C01819=1068.921,-95.321,441.532,172.288,23.007,154.216
C01820=1068.914,-95.570,441.542,172.287,23.005,154.216
C01821=1068.909,-95.820,441.552,172.285,23.004,154.216
C01822=1068.902,-96.069,441.562,172.284,23.003,154.216
C01823=1068.897,-96.318,441.573,172.282,23.001,154.216
C01824=1068.890,-96.568,441.583,172.280,23.000,154.216
C01825=1068.884,-96.818,441.594,172.279,22.999,154.216
C01826=1068.878,-97.068,441.604,172.277,22.997,154.216
C01827=1068.872,-97.318,441.614,172.275,22.996,154.216
C01828=1068.866,-97.568,441.624,172.274,22.995,154.216
C01829=1068.859,-97.850,441.635,172.272,22.993,154.215
C01830=1068.852,-98.133,441.647,172.270,22.991,154.215
C01831=1068.845,-98.416,441.659,172.268,22.990,154.215
C01832=1068.838,-98.698,441.670,172.267,22.989,154.215
C01833=1068.833,-98.948,441.681,172.265,22.987,154.215
C01834=1068.827,-99.197,441.691,172.263,22.986,154.215
C01835=1068.820,-99.447,441.701,172.261,22.985,154.215
C01836=1068.814,-99.697,441.711,172.260,22.984,154.215
C01837=1068.808,-99.947,441.722,172.258,22.982,154.215
C01838=1068.801,-100.196,441.731,172.257,22.981,154.215
C01839=1068.796,-100.446,441.742,172.255,22.980,154.215
C01840=1068.789,-100.696,441.752,172.253,22.978,154.215
C01841=1068.783,-100.945,441.761,172.252,22.977,154.215
C01842=1068.777,-101.195,441.771,172.250,22.976,154.215
C01843=1068.771,-101.445,441.782,172.248,22.975,154.215
C01844=1068.764,-101.695,441.792,172.247,22.974,154.215
C01845=1068.758,-101.944,441.802,172.245,22.972,154.215
C01846=1068.753,-102.194,441.812,172.243,22.971,154.215
C01847=1068.746,-102.444,441.822,172.242,22.970,154.215
C01848=1068.740,-102.693,441.832,172.240,22.968,154.215
C01849=1068.734,-102.943,441.843,172.238,22.968,154.216
C01850=1068.728,-103.193,441.852,172.237,22.966,154.215
C01851=1068.722,-103.443,441.862,172.235,22.965,154.215
C01852=1068.716,-103.692,441.873,172.234,22.964,154.215
C01853=1068.710,-103.942,441.882,172.232,22.962,154.215
C01854=1068.704,-104.192,441.892,172.230,22.961,154.215
C01855=1068.697,-104.441,441.902,172.228,22.960,154.216
C01856=1068.692,-104.691,441.912,172.227,22.959,154.216
C01857=1068.686,-104.941,441.922,172.225,22.958,154.216
C01858=1068.680,-105.191,441.931,172.224,22.956,154.216
C01859=1068.673,-105.440,441.942,172.222,22.956,154.216
C01860=1068.667,-105.691,441.952,172.220,22.954,154.216
C01861=1068.661,-105.940,441.962,172.219,22.953,154.216
C01862=1068.654,-106.189,441.972,172.217,22.952,154.216
C01863=1068.648,-106.439,441.982,172.215,22.951,154.216
C01864=1068.643,-106.689,441.992,172.213,22.949,154.216
C01865=1068.637,-106.939,442.001,172.212,22.948,154.216
C01866=1068.630,-107.188,442.012,172.210,22.947,154.216
C01867=1068.624,-107.438,442.021,172.208,22.946,154.216
C01868=1068.618,-107.688,442.031,172.207,22.945,154.216
C01869=1068.612,-107.938,442.041,172.205,22.943,154.216
C01870=1068.606,-108.188,442.051,172.203,22.943,154.216
C01871=1068.600,-108.437,442.061,172.202,22.941,154.216
C01872=1068.594,-108.687,442.070,172.200,22.940,154.216
C01873=1068.587,-108.937,442.080,172.198,22.939,154.216
C01874=1068.581,-109.186,442.090,172.197,22.938,154.216
C01875=1068.575,-109.436,442.099,172.195,22.937,154.216
C01876=1068.569,-109.685,442.109,172.193,22.936,154.216
C01877=1068.562,-109.935,442.119,172.191,22.935,154.216
C01878=1068.557,-110.185,442.129,172.190,22.934,154.216
C01879=1068.551,-110.435,442.139,172.188,22.932,154.216
C01880=1068.545,-110.685,442.148,172.187,22.932,154.216
C01881=1068.539,-110.935,442.158,172.186,22.931,154.216
C01882=1068.532,-111.185,442.167,172.184,22.930,154.216
C01883=1068.526,-111.434,442.178,172.182,22.929,154.216
C01884=1068.520,-111.683,442.187,172.181,22.928,154.216
C01885=1068.514,-111.933,442.197,172.179,22.926,154.216
C01886=1068.507,-112.183,442.206,172.177,22.925,154.216
C01887=1068.501,-112.433,442.216,172.175,22.924,154.216
C01888=1068.495,-112.683,442.226,172.174,22.923,154.216
C01889=1068.490,-112.933,442.236,172.172,22.922,154.217
C01890=1068.483,-113.183,442.245,172.170,22.921,154.217
C01891=1068.478,-113.432,442.254,172.169,22.920,154.217
C01892=1068.472,-113.681,442.264,172.167,22.919,154.217
C01893=1068.465,-113.962,442.275,172.165,22.918,154.217
C01894=1068.458,-114.243,442.286,172.163,22.916,154.217
C01895=1068.450,-114.522,442.296,172.161,22.916,154.217
C01896=1068.443,-114.803,442.307,172.159,22.914,154.217
C01897=1068.437,-115.053,442.317,172.157,22.913,154.217
C01898=1068.431,-115.303,442.326,172.156,22.912,154.217
C01899=1068.425,-115.552,442.336,172.154,22.911,154.217
C01900=1068.419,-115.802,442.346,172.152,22.910,154.217
C01901=1068.413,-116.052,442.355,172.151,22.909,154.217
C01902=1068.406,-116.302,442.365,172.149,22.909,154.217
C01903=1068.400,-116.552,442.374,172.147,22.907,154.217
C01904=1068.395,-116.801,442.384,172.145,22.906,154.217
C01905=1068.389,-117.050,442.393,172.144,22.906,154.218
C01906=1068.382,-117.300,442.403,172.143,22.905,154.217
C01907=1068.376,-117.550,442.412,172.141,22.904,154.218
C01908=1068.370,-117.800,442.422,172.139,22.903,154.218
C01909=1068.364,-118.050,442.431,172.138,22.902,154.218
C01910=1068.358,-118.300,442.440,172.136,22.901,154.218
C01911=1068.351,-118.550,442.449,172.134,22.900,154.218
C01912=1068.345,-118.799,442.459,172.132,22.899,154.218
C01913=1068.339,-119.049,442.468,172.131,22.898,154.218
C01914=1068.333,-119.298,442.478,172.129,22.897,154.218
C01915=1068.327,-119.548,442.487,172.127,22.896,154.218
C01916=1068.321,-119.798,442.497,172.125,22.895,154.218
C01917=1068.315,-120.048,442.506,172.124,22.895,154.218
C01918=1068.308,-120.297,442.516,172.122,22.893,154.218
C01919=1068.303,-120.548,442.525,172.120,22.893,154.218
C01920=1068.296,-120.798,442.534,172.118,22.892,154.219
C01921=1068.289,-121.047,442.543,172.117,22.890,154.219
C01922=1068.284,-121.296,442.552,172.115,22.890,154.219
C01923=1068.278,-121.546,442.562,172.113,22.889,154.219
C01924=1068.272,-121.796,442.572,172.111,22.888,154.219
C01925=1068.265,-122.046,442.581,172.110,22.887,154.219
C01926=1068.260,-122.296,442.590,172.109,22.886,154.219
C01927=1068.253,-122.546,442.599,172.107,22.886,154.219
C01928=1068.247,-122.795,442.608,172.105,22.885,154.219
C01929=1068.241,-123.044,442.618,172.103,22.884,154.219
C01930=1068.235,-123.294,442.627,172.102,22.883,154.219
C01931=1068.229,-123.545,442.636,172.100,22.882,154.219
C01932=1068.223,-123.794,442.646,172.098,22.881,154.219
C01933=1068.217,-124.044,442.655,172.096,22.880,154.220
C01934=1068.210,-124.293,442.664,172.095,22.880,154.220
C01935=1068.204,-124.543,442.673,172.093,22.879,154.220
C01936=1068.198,-124.793,442.682,172.091,22.878,154.220
C01937=1068.192,-125.043,442.692,172.089,22.877,154.220
C01938=1068.185,-125.292,442.701,172.088,22.876,154.220
C01939=1068.180,-125.542,442.709,172.086,22.875,154.220
C01940=1068.174,-125.792,442.719,172.084,22.875,154.220
C01941=1068.167,-126.042,442.728,172.083,22.874,154.220
C01942=1068.161,-126.291,442.737,172.081,22.873,154.220
C01943=1068.155,-126.542,442.746,172.079,22.873,154.221
C01944=1068.149,-126.791,442.756,172.078,22.872,154.221
C01945=1068.142,-127.040,442.764,172.076,22.871,154.221
C01946=1068.136,-127.291,442.773,172.074,22.870,154.221
C01947=1068.130,-127.540,442.783,172.072,22.870,154.221
C01948=1068.124,-127.790,442.792,172.070,22.869,154.221
C01949=1068.118,-128.041,442.801,172.069,22.868,154.221
C01950=1068.115,-128.291,442.812,172.067,22.866,154.221
C01951=1068.113,-128.542,442.822,172.066,22.863,154.221
C01952=1068.113,-128.793,442.834,172.065,22.860,154.220
C01953=1068.115,-129.046,442.847,172.064,22.856,154.220
C01954=1068.119,-129.298,442.860,172.064,22.852,154.219
C01955=1068.125,-129.549,442.875,172.064,22.847,154.218
C01956=1068.132,-129.799,442.890,172.064,22.841,154.217
C01957=1067.743,-129.822,442.718,172.016,22.987,154.250
C01958=1067.737,-129.572,442.703,172.017,22.993,154.251
C01959=1067.732,-129.320,442.688,172.017,22.997,154.252
C01960=1067.727,-129.068,442.675,172.018,23.002,154.252
C01961=1067.725,-128.816,442.662,172.018,23.005,154.253
C01962=1067.725,-128.565,442.650,172.019,23.009,154.254
C01963=1067.726,-128.314,442.639,172.020,23.011,154.254
C01964=1067.730,-128.063,442.629,172.021,23.013,154.254
C01965=1067.736,-127.812,442.619,172.023,23.014,154.254
C01966=1067.742,-127.563,442.610,172.025,23.015,154.254
C01967=1067.747,-127.313,442.601,172.027,23.015,154.254
C01968=1067.754,-127.063,442.592,172.029,23.016,154.254
C01969=1067.760,-126.814,442.583,172.030,23.017,154.253
C01970=1067.766,-126.564,442.573,172.032,23.018,154.253
C01971=1067.773,-126.314,442.564,172.034,23.018,154.253
C01972=1067.778,-126.065,442.556,172.036,23.019,154.253
C01973=1067.785,-125.815,442.546,172.037,23.021,154.253
C01974=1067.791,-125.565,442.537,172.039,23.021,154.253
C01975=1067.797,-125.315,442.528,172.040,23.022,154.253
C01976=1067.804,-125.065,442.519,172.042,23.022,154.253
C01977=1067.810,-124.815,442.509,172.044,23.023,154.253
C01978=1067.815,-124.566,442.500,172.045,23.024,154.253
C01979=1067.822,-124.316,442.492,172.047,23.025,154.252
C01980=1067.828,-124.066,442.482,172.049,23.025,154.252
C01981=1067.834,-123.816,442.473,172.051,23.027,154.252
C01982=1067.840,-123.567,442.463,172.053,23.028,154.252
C01983=1067.846,-123.317,442.455,172.054,23.028,154.252
C01984=1067.852,-123.067,442.445,172.056,23.029,154.252
C01985=1067.859,-122.818,442.436,172.058,23.030,154.252
C01986=1067.865,-122.568,442.427,172.060,23.031,154.252
C01987=1067.871,-122.318,442.417,172.061,23.032,154.252
C01988=1067.877,-122.068,442.407,172.063,23.033,154.252
C01989=1067.883,-121.819,442.399,172.065,23.033,154.252
C01990=1067.889,-121.569,442.389,172.067,23.034,154.251
C01991=1067.896,-121.319,442.380,172.068,23.035,154.251
C01992=1067.902,-121.069,442.371,172.070,23.036,154.251
C01993=1067.908,-120.820,442.361,172.071,23.037,154.251
C01994=1067.914,-120.570,442.352,172.073,23.038,154.251
C01995=1067.920,-120.319,442.343,172.075,23.039,154.251
C01996=1067.926,-120.070,442.334,172.076,23.039,154.251
C01997=1067.932,-119.821,442.324,172.078,23.040,154.251
C01998=1067.938,-119.571,442.315,172.080,23.042,154.251
C01999=1067.944,-119.321,442.305,172.082,23.042,154.251
C02000=1067.951,-119.071,442.296,172.083,23.043,154.251
C02001=1067.957,-118.822,442.286,172.085,23.044,154.251
C02002=1067.963,-118.572,442.277,172.087,23.045,154.251
C02003=1067.970,-118.322,442.267,172.089,23.046,154.251
C02004=1067.976,-118.072,442.258,172.090,23.047,154.251
C02005=1067.981,-117.823,442.249,172.092,23.048,154.250
C02006=1067.987,-117.573,442.240,172.094,23.049,154.250
C02007=1067.993,-117.323,442.230,172.095,23.050,154.250
C02008=1067.999,-117.073,442.221,172.097,23.051,154.250
C02009=1068.006,-116.823,442.211,172.099,23.052,154.250
C02010=1068.012,-116.574,442.201,172.101,23.053,154.250
C02011=1068.018,-116.324,442.192,172.103,23.054,154.250
C02012=1068.024,-116.074,442.182,172.104,23.055,154.250
C02013=1068.030,-115.824,442.173,172.106,23.056,154.250
C02014=1068.037,-115.574,442.163,172.108,23.056,154.250
C02015=1068.043,-115.325,442.154,172.109,23.058,154.250
C02016=1068.049,-115.075,442.144,172.110,23.058,154.250
C02017=1068.054,-114.826,442.135,172.112,23.059,154.250
C02018=1068.062,-114.545,442.124,172.115,23.061,154.250
C02019=1068.069,-114.265,442.113,172.116,23.062,154.250
C02020=1068.076,-113.984,442.102,172.118,23.063,154.249
C02021=1068.083,-113.703,442.092,172.120,23.064,154.250
C02022=1068.089,-113.453,442.082,172.122,23.065,154.249
C02023=1068.095,-113.205,442.072,172.123,23.066,154.249
C02024=1068.101,-112.955,442.063,172.125,23.067,154.249
C02025=1068.107,-112.705,442.053,172.127,23.068,154.249
C02026=1068.113,-112.455,442.043,172.128,23.069,154.249
C02027=1068.119,-112.205,442.033,172.130,23.070,154.249
C02028=1068.125,-111.955,442.024,172.132,23.072,154.249
C02029=1068.131,-111.706,442.014,172.133,23.072,154.249
C02030=1068.137,-111.456,442.005,172.135,23.074,154.249
C02031=1068.144,-111.206,441.995,172.137,23.074,154.249
C02032=1068.150,-110.956,441.986,172.139,23.076,154.249
C02033=1068.156,-110.707,441.975,172.140,23.076,154.249
C02034=1068.162,-110.457,441.966,172.142,23.078,154.249
C02035=1068.169,-110.207,441.956,172.144,23.079,154.249
C02036=1068.175,-109.958,441.947,172.145,23.080,154.249
C02037=1068.180,-109.707,441.937,172.147,23.081,154.249
C02038=1068.186,-109.458,441.927,172.149,23.082,154.249
C02039=1068.193,-109.208,441.917,172.150,23.083,154.249
C02040=1068.199,-108.959,441.907,172.152,23.085,154.249
C02041=1068.205,-108.709,441.898,172.154,23.085,154.249
C02042=1068.211,-108.459,441.888,172.155,23.087,154.249
C02043=1068.218,-108.209,441.878,172.157,23.087,154.249
C02044=1068.224,-107.960,441.868,172.159,23.089,154.249
C02045=1068.229,-107.710,441.858,172.161,23.090,154.249
C02046=1068.236,-107.460,441.848,172.162,23.091,154.248
C02047=1068.242,-107.210,441.839,172.164,23.092,154.248
C02048=1068.248,-106.961,441.829,172.166,23.093,154.248
C02049=1068.254,-106.711,441.819,172.167,23.094,154.248
C02050=1068.260,-106.461,441.809,172.169,23.096,154.248
C02051=1068.266,-106.212,441.799,172.171,23.097,154.248
C02052=1068.273,-105.962,441.789,172.172,23.098,154.248
C02053=1068.279,-105.713,441.779,172.174,23.099,154.248
C02054=1068.285,-105.462,441.769,172.176,23.100,154.248
C02055=1068.291,-105.212,441.759,172.177,23.102,154.248
C02056=1068.297,-104.963,441.749,172.179,23.103,154.248
C02057=1068.304,-104.713,441.739,172.181,23.104,154.248
C02058=1068.309,-104.463,441.729,172.182,23.105,154.248
C02059=1068.315,-104.214,441.719,172.184,23.106,154.248
C02060=1068.322,-103.964,441.709,172.185,23.107,154.248
C02061=1068.328,-103.714,441.700,172.186,23.109,154.248
C02062=1068.334,-103.465,441.689,172.188,23.109,154.248
C02063=1068.340,-103.215,441.679,172.190,23.111,154.248
C02064=1068.346,-102.965,441.670,172.192,23.112,154.248
C02065=1068.352,-102.715,441.659,172.193,23.113,154.248
C02066=1068.358,-102.466,441.649,172.195,23.115,154.248
C02067=1068.364,-102.216,441.640,172.196,23.116,154.248
C02068=1068.370,-101.967,441.630,172.198,23.117,154.248
C02069=1068.376,-101.717,441.619,172.200,23.118,154.248
C02070=1068.383,-101.467,441.609,172.201,23.119,154.248
C02071=1068.389,-101.217,441.599,172.203,23.121,154.248
C02072=1068.395,-100.967,441.589,172.205,23.122,154.248
C02073=1068.401,-100.718,441.579,172.206,23.123,154.248
C02074=1068.407,-100.468,441.569,172.208,23.125,154.248
C02075=1068.413,-100.218,441.558,172.210,23.126,154.248
C02076=1068.419,-99.969,441.549,172.211,23.127,154.248
C02077=1068.426,-99.719,441.538,172.213,23.128,154.248
C02078=1068.432,-99.469,441.528,172.215,23.129,154.248
C02079=1068.438,-99.219,441.518,172.216,23.131,154.248
C02080=1068.444,-98.970,441.508,172.218,23.132,154.248
C02081=1068.450,-98.719,441.498,172.220,23.133,154.248
C02082=1068.457,-98.436,441.486,172.222,23.135,154.248
C02083=1068.464,-98.154,441.475,172.224,23.136,154.248
C02084=1068.471,-97.871,441.463,172.225,23.138,154.248
C02085=1068.477,-97.589,441.452,172.227,23.139,154.248
C02086=1068.484,-97.339,441.441,172.230,23.141,154.248
C02087=1068.490,-97.089,441.431,172.231,23.142,154.248
C02088=1068.496,-96.840,441.421,172.233,23.143,154.248
C02089=1068.502,-96.590,441.410,172.234,23.145,154.248
C02090=1068.508,-96.341,441.400,172.236,23.147,154.248
C02091=1068.514,-96.091,441.389,172.238,23.148,154.248
C02092=1068.520,-95.841,441.380,172.239,23.149,154.248
C02093=1068.526,-95.592,441.369,172.241,23.150,154.248
C02094=1068.532,-95.341,441.359,172.242,23.152,154.248
C02095=1068.538,-95.092,441.348,172.244,23.153,154.249
C02096=1068.544,-94.842,441.337,172.246,23.154,154.249
C02097=1068.550,-94.592,441.328,172.247,23.156,154.249
C02098=1068.556,-94.343,441.317,172.249,23.157,154.249
C02099=1068.562,-94.093,441.307,172.250,23.159,154.249
C02100=1068.568,-93.844,441.296,172.252,23.160,154.249
C02101=1068.575,-93.594,441.286,172.254,23.162,154.249
C02102=1068.580,-93.344,441.276,172.255,23.163,154.249
C02103=1068.586,-93.094,441.265,172.257,23.164,154.249
C02104=1068.592,-92.844,441.255,172.259,23.166,154.249
C02105=1068.598,-92.595,441.244,172.260,23.167,154.249
C02106=1068.605,-92.345,441.234,172.262,23.169,154.249
C02107=1068.611,-92.095,441.224,172.263,23.170,154.249
C02108=1068.616,-91.845,441.213,172.265,23.171,154.249
C02109=1068.623,-91.596,441.202,172.267,23.173,154.249
C02110=1068.629,-91.347,441.191,172.268,23.174,154.249
C02111=1068.635,-91.096,441.182,172.270,23.176,154.249
C02112=1068.641,-90.847,441.171,172.271,23.177,154.249
C02113=1068.647,-90.597,441.160,172.273,23.179,154.249
C02114=1068.653,-90.347,441.150,172.275,23.180,154.249
C02115=1068.659,-90.098,441.139,172.276,23.181,154.249
C02116=1068.666,-89.848,441.129,172.278,23.183,154.249
C02117=1068.671,-89.599,441.118,172.279,23.184,154.249
C02118=1068.677,-89.349,441.108,172.281,23.186,154.249
C02119=1068.683,-89.099,441.097,172.283,23.187,154.249
C02120=1068.690,-88.849,441.086,172.284,23.189,154.250
C02121=1068.696,-88.600,441.076,172.286,23.190,154.250
C02122=1068.702,-88.350,441.066,172.287,23.192,154.250
C02123=1068.707,-88.100,441.055,172.289,23.193,154.250
C02124=1068.714,-87.850,441.044,172.290,23.195,154.250
C02125=1068.720,-87.601,441.033,172.292,23.196,154.250
C02126=1068.726,-87.352,441.022,172.294,23.197,154.250
C02127=1068.733,-87.101,441.012,172.295,23.199,154.250
C02128=1068.738,-86.852,441.002,172.297,23.201,154.250
C02129=1068.744,-86.602,440.991,172.298,23.202,154.250
C02130=1068.751,-86.353,440.980,172.300,23.203,154.250
C02131=1068.757,-86.103,440.969,172.301,23.205,154.250
C02132=1068.762,-85.853,440.959,172.303,23.206,154.250
C02133=1068.769,-85.603,440.949,172.305,23.208,154.250
C02134=1068.775,-85.353,440.938,172.306,23.209,154.250
C02135=1068.781,-85.104,440.927,172.308,23.211,154.250
C02136=1068.787,-84.855,440.916,172.309,23.212,154.250
C02137=1068.794,-84.604,440.905,172.311,23.214,154.250
C02138=1068.800,-84.355,440.894,172.313,23.215,154.250
C02139=1068.806,-84.106,440.884,172.314,23.217,154.250
C02140=1068.812,-83.855,440.873,172.316,23.218,154.251
C02141=1068.818,-83.605,440.863,172.317,23.220,154.251
C02142=1068.824,-83.356,440.852,172.320,23.222,154.251
C02143=1068.831,-83.106,440.841,172.321,23.223,154.251
C02144=1068.836,-82.856,440.830,172.323,23.225,154.251
C02145=1068.843,-82.607,440.820,172.325,23.226,154.251
C02146=1068.850,-82.326,440.807,172.326,23.228,154.251
C02147=1068.857,-82.046,440.795,172.328,23.229,154.251
C02148=1068.864,-81.766,440.783,172.329,23.231,154.251
C02149=1068.871,-81.486,440.771,172.332,23.233,154.251
C02150=1068.877,-81.235,440.759,172.333,23.235,154.251
C02151=1068.883,-80.986,440.749,172.335,23.236,154.251
C02152=1068.889,-80.737,440.738,172.336,23.238,154.251
C02153=1068.895,-80.487,440.727,172.338,23.239,154.251
C02154=1068.902,-80.237,440.717,172.339,23.241,154.251
C02155=1068.908,-79.987,440.705,172.341,23.243,154.252
C02156=1068.914,-79.738,440.694,172.343,23.244,154.252
C02157=1068.920,-79.488,440.684,172.344,23.246,154.252
C02158=1068.926,-79.238,440.672,172.346,23.247,154.252
C02159=1068.932,-78.989,440.661,172.347,23.249,154.252
C02160=1068.938,-78.739,440.651,172.349,23.250,154.252
C02161=1068.945,-78.489,440.640,172.350,23.252,154.252
C02162=1068.950,-78.240,440.629,172.352,23.254,154.252
C02163=1068.957,-77.990,440.618,172.353,23.255,154.252
C02164=1068.962,-77.740,440.607,172.355,23.257,154.252
C02165=1068.968,-77.491,440.596,172.356,23.259,154.252
C02166=1068.975,-77.240,440.585,172.358,23.260,154.253
C02167=1068.980,-76.991,440.574,172.360,23.262,154.253
C02168=1068.986,-76.741,440.563,172.361,23.264,154.253
C02169=1068.993,-76.492,440.551,172.363,23.266,154.253
C02170=1068.998,-76.242,440.540,172.365,23.267,154.253
C02171=1069.005,-75.992,440.529,172.366,23.269,154.253
C02172=1069.010,-75.743,440.518,172.368,23.270,154.253
C02173=1069.017,-75.492,440.507,172.370,23.272,154.253
C02174=1069.023,-75.243,440.497,172.371,23.274,154.253
C02175=1069.029,-74.994,440.486,172.373,23.275,154.253
C02176=1069.036,-74.744,440.474,172.374,23.277,154.253
C02177=1069.041,-74.495,440.463,172.376,23.279,154.253
C02178=1069.048,-74.245,440.452,172.377,23.281,154.254
C02179=1069.054,-73.995,440.441,172.379,23.282,154.254
C02180=1069.060,-73.745,440.430,172.380,23.284,154.254
C02181=1069.066,-73.496,440.418,172.382,23.286,154.254
C02182=1069.071,-73.246,440.406,172.383,23.287,154.254
C02183=1069.077,-72.996,440.395,172.385,23.289,154.254
C02184=1069.083,-72.747,440.384,172.386,23.291,154.254
C02185=1069.089,-72.496,440.373,172.388,23.293,154.254
C02186=1069.095,-72.247,440.362,172.389,23.294,154.254
C02187=1069.101,-71.998,440.351,172.391,23.296,154.255
C02188=1069.107,-71.747,440.339,172.392,23.298,154.255
C02189=1069.112,-71.498,440.328,172.394,23.299,154.255
C02190=1069.119,-71.248,440.316,172.395,23.301,154.255
C02191=1069.125,-70.999,440.305,172.397,23.303,154.255
C02192=1069.131,-70.749,440.294,172.399,23.305,154.255
C02193=1069.137,-70.500,440.282,172.401,23.307,154.255
C02194=1069.142,-70.250,440.271,172.402,23.309,154.255
C02195=1069.149,-70.000,440.260,172.404,23.311,154.255
C02196=1069.155,-69.751,440.248,172.405,23.312,154.256
C02197=1069.161,-69.501,440.237,172.407,23.314,154.256
C02198=1069.167,-69.251,440.226,172.408,23.316,154.256
C02199=1069.173,-69.002,440.214,172.410,23.318,154.256
C02200=1069.178,-68.752,440.202,172.411,23.320,154.256
C02201=1069.185,-68.502,440.191,172.413,23.321,154.256
C02202=1069.191,-68.253,440.180,172.414,23.323,154.256
C02203=1069.197,-68.003,440.168,172.416,23.325,154.256
C02204=1069.203,-67.753,440.157,172.417,23.327,154.257
C02205=1069.209,-67.503,440.145,172.419,23.329,154.257
C02206=1069.214,-67.254,440.134,172.420,23.331,154.257
C02207=1069.221,-67.004,440.122,172.421,23.333,154.257
C02208=1069.227,-66.755,440.111,172.423,23.334,154.257
C02209=1069.232,-66.504,440.099,172.425,23.336,154.257
C02210=1069.239,-66.227,440.087,172.427,23.339,154.257
C02211=1069.246,-65.949,440.073,172.428,23.340,154.258
C02212=1069.253,-65.670,440.061,172.430,23.342,154.258
C02213=1069.259,-65.392,440.048,172.432,23.345,154.258
C02214=1069.265,-65.142,440.037,172.434,23.346,154.258
C02215=1069.272,-64.893,440.025,172.435,23.348,154.258
C02216=1069.278,-64.643,440.014,172.436,23.350,154.258
C02217=1069.283,-64.393,440.002,172.438,23.352,154.258
C02218=1069.289,-64.144,439.991,172.440,23.353,154.258
C02219=1069.296,-63.894,439.979,172.441,23.355,154.259
C02220=1069.302,-63.645,439.968,172.443,23.357,154.259
C02221=1069.307,-63.395,439.955,172.444,23.359,154.259
C02222=1069.314,-63.145,439.944,172.445,23.361,154.259
C02223=1069.320,-62.896,439.932,172.447,23.363,154.259
C02224=1069.326,-62.645,439.921,172.448,23.365,154.259
C02225=1069.332,-62.396,439.909,172.450,23.366,154.259
C02226=1069.338,-62.146,439.898,172.451,23.368,154.260
C02227=1069.345,-61.897,439.886,172.453,23.370,154.260
C02228=1069.350,-61.647,439.874,172.454,23.372,154.260
C02229=1069.356,-61.397,439.862,172.456,23.374,154.260
C02230=1069.362,-61.148,439.851,172.458,23.376,154.260
C02231=1069.369,-60.898,439.840,172.460,23.378,154.260
C02232=1069.374,-60.648,439.827,172.461,23.380,154.260
C02233=1069.380,-60.399,439.816,172.463,23.382,154.261
C02234=1069.387,-60.149,439.804,172.464,23.384,154.261
C02235=1069.392,-59.900,439.792,172.465,23.386,154.261
C02236=1069.398,-59.650,439.781,172.467,23.387,154.261
C02237=1069.405,-59.400,439.769,172.468,23.389,154.261
C02238=1069.411,-59.151,439.758,172.470,23.391,154.261
C02239=1069.417,-58.901,439.745,172.471,23.393,154.261
C02240=1069.423,-58.651,439.733,172.473,23.395,154.262
C02241=1069.429,-58.402,439.722,172.474,23.397,154.262
C02242=1069.435,-58.152,439.710,172.476,23.399,154.262
C02243=1069.442,-57.902,439.698,172.477,23.400,154.262
C02244=1069.447,-57.653,439.687,172.479,23.402,154.262
C02245=1069.453,-57.403,439.675,172.480,23.404,154.262
C02246=1069.460,-57.153,439.663,172.482,23.406,154.263
C02247=1069.466,-56.904,439.652,172.484,23.408,154.263
C02248=1069.472,-56.654,439.639,172.485,23.410,154.263
C02249=1069.478,-56.404,439.627,172.487,23.412,154.263
C02250=1069.485,-56.155,439.615,172.488,23.414,154.263
C02251=1069.490,-55.905,439.604,172.490,23.416,154.263
C02252=1069.497,-55.655,439.592,172.491,23.418,154.263
C02253=1069.503,-55.406,439.580,172.493,23.420,154.263
C02254=1069.509,-55.157,439.568,172.494,23.421,154.264
C02255=1069.515,-54.907,439.556,172.496,23.423,154.264
C02256=1069.522,-54.657,439.544,172.497,23.425,154.264
C02257=1069.527,-54.407,439.532,172.499,23.428,154.264
C02258=1069.534,-54.158,439.520,172.500,23.429,154.264
C02259=1069.540,-53.908,439.509,172.502,23.431,154.264
C02260=1069.546,-53.658,439.496,172.503,23.433,154.265
C02261=1069.552,-53.409,439.485,172.504,23.435,154.265
C02262=1069.558,-53.160,439.473,172.507,23.437,154.265
C02263=1069.564,-52.910,439.460,172.508,23.439,154.265
C02264=1069.571,-52.660,439.449,172.510,23.441,154.265
C02265=1069.577,-52.410,439.437,172.511,23.443,154.265
C02266=1069.583,-52.161,439.425,172.513,23.445,154.265
C02267=1069.589,-51.911,439.413,172.514,23.447,154.266
C02268=1069.595,-51.661,439.400,172.516,23.449,154.266
C02269=1069.602,-51.412,439.389,172.517,23.451,154.266
C02270=1069.608,-51.162,439.376,172.518,23.453,154.266
C02271=1069.613,-50.912,439.365,172.520,23.455,154.266
C02272=1069.620,-50.663,439.353,172.521,23.457,154.266
C02273=1069.626,-50.413,439.341,172.523,23.458,154.267
C02274=1069.633,-50.136,439.327,172.525,23.461,154.267
C02275=1069.639,-49.859,439.314,172.527,23.463,154.267
C02276=1069.646,-49.583,439.300,172.528,23.466,154.267
C02277=1069.653,-49.306,439.287,172.529,23.467,154.267
C02278=1069.659,-49.056,439.274,172.532,23.470,154.268
C02279=1069.665,-48.806,439.262,172.533,23.472,154.268
C02280=1069.671,-48.557,439.250,172.534,23.474,154.268
C02281=1069.677,-48.307,439.237,172.536,23.476,154.268
C02282=1069.683,-48.058,439.225,172.537,23.478,154.268
C02283=1069.689,-47.808,439.213,172.539,23.480,154.269
C02284=1069.694,-47.558,439.201,172.540,23.483,154.269
C02285=1069.701,-47.309,439.189,172.542,23.484,154.269
C02286=1069.707,-47.059,439.176,172.543,23.486,154.269
C02287=1069.713,-46.809,439.164,172.544,23.489,154.269
C02288=1069.719,-46.560,439.152,172.546,23.491,154.270
C02289=1069.725,-46.310,439.139,172.547,23.492,154.270
C02290=1069.731,-46.060,439.127,172.549,23.495,154.270
C02291=1069.737,-45.811,439.115,172.550,23.497,154.270
C02292=1069.743,-45.561,439.102,172.552,23.499,154.270
C02293=1069.749,-45.312,439.090,172.554,23.501,154.270
C02294=1069.755,-45.062,439.078,172.555,23.503,154.271
C02295=1069.761,-44.812,439.066,172.557,23.505,154.271
C02296=1069.767,-44.562,439.053,172.558,23.508,154.271
C02297=1069.773,-44.313,439.041,172.559,23.509,154.271
C02298=1069.779,-44.064,439.029,172.561,23.512,154.271
C02299=1069.785,-43.814,439.016,172.562,23.514,154.272
C02300=1069.791,-43.564,439.004,172.564,23.516,154.272
C02301=1069.797,-43.314,438.991,172.565,23.518,154.272
C02302=1069.803,-43.065,438.979,172.567,23.520,154.272
C02303=1069.810,-42.815,438.966,172.568,23.522,154.272
C02304=1069.815,-42.566,438.954,172.569,23.524,154.273
C02305=1069.821,-42.316,438.941,172.571,23.526,154.273
C02306=1069.827,-42.067,438.929,172.572,23.528,154.273
C02307=1069.833,-41.817,438.917,172.574,23.531,154.273
C02308=1069.839,-41.567,438.904,172.576,23.533,154.273
C02309=1069.846,-41.317,438.892,172.577,23.535,154.274
C02310=1069.852,-41.068,438.879,172.579,23.537,154.274
C02311=1069.858,-40.818,438.866,172.580,23.539,154.274
C02312=1069.863,-40.569,438.854,172.582,23.541,154.274
C02313=1069.870,-40.319,438.842,172.583,23.543,154.274
C02314=1069.876,-40.069,438.830,172.584,23.545,154.275
C02315=1069.882,-39.820,438.816,172.586,23.547,154.275
C02316=1069.888,-39.570,438.804,172.587,23.550,154.275
C02317=1069.894,-39.320,438.791,172.589,23.552,154.275
C02318=1069.901,-39.071,438.779,172.590,23.554,154.275
C02319=1069.907,-38.821,438.767,172.591,23.556,154.276
C02320=1069.913,-38.572,438.754,172.593,23.558,154.276
C02321=1069.919,-38.322,438.741,172.595,23.560,154.276
C02322=1069.924,-38.073,438.729,172.596,23.563,154.276
C02323=1069.930,-37.823,438.716,172.598,23.565,154.276
C02324=1069.936,-37.574,438.703,172.599,23.567,154.277
C02325=1069.942,-37.324,438.690,172.601,23.569,154.277
C02326=1069.948,-37.074,438.678,172.602,23.571,154.277
C02327=1069.954,-36.825,438.665,172.603,23.573,154.277
C02328=1069.961,-36.575,438.653,172.605,23.576,154.277
C02329=1069.967,-36.325,438.640,172.606,23.578,154.278
C02330=1069.973,-36.076,438.627,172.608,23.580,154.278
C02331=1069.978,-35.827,438.615,172.609,23.582,154.278
C02332=1069.984,-35.577,438.602,172.610,23.584,154.278
C02333=1069.990,-35.327,438.589,172.612,23.587,154.279
C02334=1069.996,-35.078,438.576,172.613,23.589,154.279
C02335=1070.002,-34.828,438.564,172.615,23.591,154.279
C02336=1070.008,-34.578,438.550,172.617,23.594,154.279
C02337=1070.014,-34.329,438.538,172.618,23.596,154.279
C02338=1070.021,-34.052,438.523,172.619,23.598,154.280
C02339=1070.027,-33.775,438.510,172.621,23.601,154.280
C02340=1070.034,-33.499,438.495,172.623,23.603,154.280
C02341=1070.040,-33.222,438.481,172.624,23.606,154.280
C02342=1070.046,-32.973,438.468,172.626,23.608,154.281
C02343=1070.053,-32.723,438.455,172.627,23.610,154.281
C02344=1070.058,-32.473,438.442,172.629,23.612,154.281
C02345=1070.064,-32.223,438.430,172.630,23.614,154.281
C02346=1070.071,-31.974,438.416,172.631,23.617,154.282
C02347=1070.076,-31.724,438.404,172.633,23.619,154.282
C02348=1070.083,-31.475,438.391,172.634,23.621,154.282
C02349=1070.089,-31.225,438.378,172.635,23.623,154.282
C02350=1070.095,-30.976,438.365,172.638,23.626,154.282
C02351=1070.101,-30.726,438.352,172.639,23.628,154.283
C02352=1070.107,-30.477,438.339,172.641,23.630,154.283
C02353=1070.113,-30.227,438.326,172.642,23.632,154.283
C02354=1070.119,-29.978,438.313,172.643,23.635,154.283
C02355=1070.125,-29.728,438.301,172.645,23.637,154.283
C02356=1070.131,-29.479,438.287,172.646,23.639,154.284
C02357=1070.137,-29.229,438.275,172.647,23.641,154.284
C02358=1070.143,-28.979,438.261,172.649,23.643,154.284
C02359=1070.149,-28.729,438.249,172.650,23.646,154.284
C02360=1070.155,-28.480,438.236,172.652,23.648,154.285
C02361=1070.161,-28.230,438.223,172.653,23.650,154.285
C02362=1070.168,-27.981,438.210,172.654,23.652,154.285
C02363=1070.174,-27.732,438.197,172.657,23.655,154.285
C02364=1070.180,-27.482,438.184,172.658,23.657,154.286
C02365=1070.186,-27.232,438.170,172.659,23.659,154.286
C02366=1070.192,-26.982,438.158,172.661,23.661,154.286
C02367=1070.198,-26.732,438.144,172.662,23.664,154.286
C02368=1070.204,-26.483,438.131,172.663,23.666,154.287
C02369=1070.210,-26.233,438.118,172.665,23.669,154.287
C02370=1070.216,-25.984,438.105,172.666,23.670,154.287
C02371=1070.221,-25.734,438.092,172.668,23.673,154.287
C02372=1070.228,-25.485,438.078,172.669,23.675,154.287
C02373=1070.234,-25.235,438.065,172.670,23.678,154.288
C02374=1070.240,-24.985,438.053,172.672,23.680,154.288
C02375=1070.245,-24.736,438.039,172.673,23.682,154.288
C02376=1070.251,-24.487,438.025,172.675,23.685,154.288
C02377=1070.257,-24.237,438.013,172.677,23.687,154.289
C02378=1070.264,-23.987,438.000,172.678,23.690,154.289
C02379=1070.269,-23.738,437.986,172.679,23.691,154.289
C02380=1070.275,-23.489,437.973,172.681,23.694,154.289
C02381=1070.281,-23.239,437.960,172.682,23.696,154.290
C02382=1070.287,-22.989,437.946,172.683,23.699,154.290
C02383=1070.293,-22.740,437.933,172.685,23.701,154.290
C02384=1070.299,-22.489,437.920,172.686,23.703,154.290
C02385=1070.306,-22.240,437.907,172.687,23.705,154.291
C02386=1070.311,-21.990,437.893,172.689,23.708,154.291
C02387=1070.317,-21.741,437.879,172.690,23.710,154.291
C02388=1070.323,-21.491,437.867,172.691,23.713,154.291
C02389=1070.329,-21.242,437.853,172.694,23.715,154.292
C02390=1070.335,-20.993,437.840,172.695,23.717,154.292
C02391=1070.341,-20.743,437.827,172.696,23.720,154.292
C02392=1070.347,-20.494,437.813,172.698,23.722,154.292
C02393=1070.353,-20.243,437.800,172.699,23.724,154.293
C02394=1070.359,-19.994,437.786,172.700,23.727,154.293
C02395=1070.365,-19.745,437.773,172.702,23.729,154.293
C02396=1070.371,-19.495,437.759,172.703,23.731,154.293
C02397=1070.377,-19.246,437.746,172.705,23.733,154.294
C02398=1070.383,-18.996,437.733,172.706,23.736,154.294
C02399=1070.389,-18.746,437.720,172.707,23.738,154.294
C02400=1070.395,-18.496,437.706,172.709,23.741,154.295
C02401=1070.402,-18.247,437.693,172.710,23.743,154.295
C02402=1070.408,-17.970,437.677,172.712,23.745,154.295
C02403=1070.415,-17.693,437.662,172.713,23.748,154.295
C02404=1070.421,-17.415,437.648,172.715,23.751,154.296
C02405=1070.428,-17.138,437.633,172.717,23.754,154.296
C02406=1070.434,-16.888,437.619,172.718,23.756,154.296
C02407=1070.440,-16.639,437.606,172.720,23.758,154.296
C02408=1070.447,-16.389,437.592,172.721,23.760,154.297
C02409=1070.452,-16.140,437.578,172.722,23.763,154.297
C02410=1070.458,-15.890,437.565,172.724,23.765,154.297
C02411=1070.465,-15.641,437.552,172.725,23.767,154.297
C02412=1070.471,-15.391,437.538,172.726,23.770,154.298
C02413=1070.476,-15.141,437.525,172.728,23.772,154.298
C02414=1070.482,-14.891,437.511,172.729,23.775,154.298
C02415=1070.488,-14.642,437.498,172.730,23.777,154.298
C02416=1070.494,-14.392,437.484,172.732,23.779,154.299
C02417=1070.500,-14.143,437.471,172.734,23.782,154.299
C02418=1070.506,-13.893,437.457,172.735,23.784,154.299
C02419=1070.512,-13.644,437.443,172.737,23.786,154.299
C02420=1070.518,-13.394,437.430,172.738,23.789,154.300
C02421=1070.523,-13.145,437.416,172.739,23.791,154.300
C02422=1070.530,-12.895,437.402,172.741,23.794,154.300
C02423=1070.535,-12.645,437.388,172.742,23.796,154.301
C02424=1070.542,-12.396,437.375,172.743,23.799,154.301
C02425=1070.547,-12.147,437.360,172.745,23.801,154.301
C02426=1070.554,-11.897,437.347,172.746,23.803,154.301
C02427=1070.560,-11.647,437.333,172.747,23.806,154.302
C02428=1070.566,-11.398,437.320,172.749,23.808,154.302
C02429=1070.571,-11.149,437.306,172.750,23.811,154.302
C02430=1070.577,-10.899,437.292,172.752,23.813,154.302
C02431=1070.584,-10.649,437.278,172.754,23.816,154.303
C02432=1070.589,-10.399,437.264,172.755,23.818,154.303
C02433=1070.595,-10.150,437.251,172.756,23.821,154.303
C02434=1070.601,-9.901,437.237,172.758,23.823,154.304
C02435=1070.607,-9.650,437.223,172.759,23.825,154.304
C02436=1070.613,-9.402,437.209,172.760,23.828,154.304
C02437=1070.619,-9.152,437.195,172.762,23.830,154.304
C02438=1070.625,-8.903,437.182,172.763,23.833,154.305
C02439=1070.631,-8.653,437.168,172.764,23.835,154.305
C02440=1070.637,-8.403,437.154,172.766,23.837,154.305
C02441=1070.643,-8.154,437.140,172.767,23.840,154.305
C02442=1070.649,-7.904,437.126,172.768,23.842,154.306
C02443=1070.655,-7.655,437.112,172.771,23.845,154.306
C02444=1070.661,-7.405,437.098,172.772,23.847,154.306
C02445=1070.667,-7.155,437.084,172.773,23.850,154.307
C02446=1070.673,-6.906,437.071,172.775,23.852,154.307
C02447=1070.679,-6.657,437.056,172.776,23.855,154.307
C02448=1070.685,-6.407,437.043,172.777,23.857,154.307
C02449=1070.691,-6.157,437.029,172.779,23.859,154.308
C02450=1070.697,-5.908,437.015,172.780,23.862,154.308
C02451=1070.703,-5.659,437.001,172.781,23.864,154.308
C02452=1070.709,-5.409,436.987,172.783,23.867,154.308
C02453=1070.715,-5.159,436.973,172.784,23.869,154.309
C02454=1070.721,-4.910,436.960,172.785,23.871,154.309
C02455=1070.727,-4.660,436.945,172.787,23.874,154.309
C02456=1070.733,-4.411,436.931,172.789,23.877,154.310
C02457=1070.740,-4.161,436.917,172.790,23.879,154.310
C02458=1070.745,-3.911,436.903,172.791,23.881,154.310
C02459=1070.751,-3.662,436.889,172.793,23.884,154.310
C02460=1070.758,-3.412,436.875,172.794,23.886,154.311
C02461=1070.763,-3.163,436.861,172.795,23.889,154.311
C02462=1070.769,-2.914,436.847,172.797,23.891,154.311
C02463=1070.775,-2.663,436.832,172.798,23.893,154.311
C02464=1070.781,-2.414,436.819,172.799,23.896,154.312
C02465=1070.787,-2.165,436.805,172.801,23.899,154.312
C02466=1070.793,-1.886,436.789,172.803,23.901,154.312
C02467=1070.800,-1.606,436.773,172.804,23.904,154.313
C02468=1070.806,-1.328,436.756,172.805,23.907,154.313
C02469=1070.813,-1.049,436.741,172.807,23.910,154.313
C02470=1070.819,-0.799,436.726,172.809,23.913,154.314
C02471=1070.825,-0.550,436.712,172.810,23.915,154.314
C02472=1070.830,-0.300,436.699,172.811,23.917,154.314
C02473=1070.837,-0.051,436.684,172.813,23.920,154.315
C02474=1070.842,0.199,436.670,172.814,23.923,154.315
C02475=1070.848,0.448,436.655,172.815,23.925,154.315
C02476=1070.854,0.698,436.641,172.817,23.928,154.316
C02477=1070.860,0.947,436.626,172.818,23.930,154.316
C02478=1070.867,1.197,436.613,172.819,23.932,154.316
C02479=1070.872,1.447,436.599,172.821,23.935,154.316
C02480=1070.878,1.696,436.584,172.822,23.938,154.317
C02481=1070.884,1.946,436.570,172.823,23.940,154.317
C02482=1070.890,2.195,436.555,172.825,23.942,154.317
C02483=1070.895,2.444,436.542,172.827,23.945,154.318
C02484=1070.902,2.694,436.527,172.828,23.948,154.318
C02485=1070.907,2.944,436.513,172.829,23.951,154.318
C02486=1070.913,3.193,436.498,172.831,23.953,154.319
C02487=1070.919,3.442,436.483,172.832,23.955,154.319
C02488=1070.925,3.692,436.469,172.833,23.958,154.319
C02489=1070.931,3.941,436.454,172.835,23.960,154.319
C02490=1070.937,4.191,436.441,172.836,23.963,154.320
C02491=1070.943,4.441,436.426,172.837,23.965,154.320
C02492=1070.948,4.690,436.412,172.839,23.968,154.320
C02493=1070.955,4.940,436.397,172.840,23.970,154.321
C02494=1070.960,5.190,436.383,172.841,23.973,154.321
C02495=1070.967,5.439,436.368,172.843,23.975,154.321
C02496=1070.972,5.688,436.353,172.845,23.978,154.321
C02497=1070.978,5.938,436.340,172.846,23.981,154.322
C02498=1070.984,6.187,436.325,172.847,23.983,154.322
C02499=1070.990,6.437,436.311,172.849,23.986,154.322
C02500=1070.996,6.687,436.296,172.850,23.988,154.323
C02501=1071.002,6.936,436.281,172.851,23.990,154.323
C02502=1071.008,7.186,436.267,172.853,23.993,154.323
C02503=1071.014,7.435,436.252,172.854,23.996,154.324
C02504=1071.020,7.684,436.237,172.855,23.998,154.324
C02505=1071.026,7.934,436.224,172.857,24.000,154.324
C02506=1071.032,8.184,436.209,172.858,24.003,154.324
C02507=1071.038,8.433,436.194,172.859,24.005,154.325
C02508=1071.044,8.683,436.180,172.860,24.008,154.325
C02509=1071.050,8.932,436.165,172.863,24.011,154.325
C02510=1071.056,9.181,436.150,172.864,24.013,154.326
C02511=1071.062,9.430,436.136,172.865,24.016,154.326
C02512=1071.068,9.681,436.121,172.867,24.018,154.326
C02513=1071.074,9.930,436.107,172.868,24.021,154.326
C02514=1071.080,10.179,436.092,172.869,24.024,154.327
C02515=1071.086,10.429,436.078,172.871,24.026,154.327
C02516=1071.092,10.679,436.063,172.872,24.028,154.327
C02517=1071.098,10.928,436.048,172.873,24.031,154.328
C02518=1071.104,11.177,436.034,172.875,24.033,154.328
C02519=1071.110,11.427,436.019,172.876,24.035,154.328
C02520=1071.116,11.676,436.005,172.877,24.038,154.329
C02521=1071.122,11.926,435.990,172.879,24.041,154.329
C02522=1071.128,12.175,435.975,172.881,24.044,154.329
C02523=1071.134,12.425,435.960,172.882,24.046,154.329
C02524=1071.141,12.674,435.945,172.884,24.048,154.330
C02525=1071.146,12.924,435.932,172.885,24.051,154.330
C02526=1071.153,13.174,435.917,172.886,24.054,154.330
C02527=1071.159,13.423,435.902,172.887,24.056,154.331
C02528=1071.165,13.672,435.887,172.889,24.058,154.331
C02529=1071.171,13.922,435.872,172.890,24.061,154.331
C02530=1071.177,14.203,435.856,172.891,24.064,154.332
C02531=1071.184,14.484,435.839,172.894,24.067,154.332
C02532=1071.191,14.765,435.822,172.895,24.069,154.332
C02533=1071.198,15.045,435.805,172.896,24.072,154.333
C02534=1071.203,15.295,435.791,172.898,24.075,154.333
C02535=1071.209,15.545,435.776,172.900,24.078,154.333
C02536=1071.215,15.795,435.761,172.901,24.081,154.334
C02537=1071.221,16.044,435.746,172.902,24.083,154.334
C02538=1071.227,16.293,435.731,172.903,24.085,154.334
C02539=1071.232,16.542,435.716,172.905,24.088,154.335
C02540=1071.239,16.792,435.701,172.906,24.091,154.335
C02541=1071.245,17.042,435.686,172.907,24.093,154.335
C02542=1071.250,17.291,435.671,172.909,24.095,154.335
C02543=1071.257,17.541,435.656,172.910,24.098,154.336
C02544=1071.262,17.790,435.642,172.911,24.101,154.336
C02545=1071.269,18.039,435.627,172.913,24.103,154.336
C02546=1071.274,18.289,435.611,172.915,24.106,154.337
C02547=1071.280,18.538,435.597,172.916,24.109,154.337
C02548=1071.287,18.788,435.582,172.917,24.111,154.337
C02549=1071.292,19.037,435.566,172.919,24.114,154.338
C02550=1071.298,19.287,435.551,172.920,24.117,154.338
C02551=1071.304,19.536,435.537,172.921,24.119,154.338
C02552=1071.309,19.786,435.521,172.923,24.121,154.339
C02553=1071.316,20.035,435.506,172.924,24.124,154.339
C02554=1071.322,20.285,435.491,172.925,24.127,154.339
C02555=1071.327,20.534,435.476,172.927,24.129,154.340
C02556=1071.334,20.784,435.461,172.928,24.131,154.340
C02557=1071.340,21.034,435.446,172.929,24.134,154.340
C02558=1071.345,21.283,435.431,172.931,24.137,154.340
C02559=1071.351,21.533,435.416,172.933,24.139,154.341
C02560=1071.357,21.782,435.400,172.934,24.142,154.341
C02561=1071.363,22.031,435.385,172.935,24.145,154.341
C02562=1071.370,22.280,435.370,172.937,24.147,154.342
C02563=1071.375,22.530,435.355,172.938,24.150,154.342
C02564=1071.381,22.779,435.340,172.939,24.152,154.342
C02565=1071.387,23.029,435.325,172.941,24.155,154.343
C02566=1071.392,23.278,435.310,172.942,24.158,154.343
C02567=1071.398,23.528,435.294,172.943,24.160,154.343
C02568=1071.405,23.777,435.279,172.944,24.163,154.344
C02569=1071.411,24.027,435.264,172.946,24.166,154.344
C02570=1071.416,24.276,435.249,172.947,24.168,154.344
C02571=1071.423,24.526,435.234,172.949,24.171,154.345
C02572=1071.428,24.776,435.218,172.950,24.174,154.345
C02573=1071.434,25.024,435.203,172.952,24.176,154.345
C02574=1071.440,25.274,435.188,172.953,24.178,154.346
C02575=1071.446,25.524,435.173,172.954,24.181,154.346
C02576=1071.451,25.773,435.157,172.956,24.184,154.346
C02577=1071.458,26.022,435.142,172.957,24.186,154.347
C02578=1071.464,26.272,435.126,172.958,24.189,154.347
C02579=1071.470,26.522,435.111,172.960,24.191,154.347
C02580=1071.476,26.771,435.097,172.961,24.194,154.348
C02581=1071.482,27.020,435.080,172.962,24.197,154.348
C02582=1071.487,27.270,435.065,172.964,24.199,154.348
C02583=1071.494,27.520,435.050,172.966,24.202,154.348
C02584=1071.499,27.769,435.035,172.967,24.205,154.349
C02585=1071.506,28.018,435.019,172.968,24.207,154.349
C02586=1071.511,28.268,435.004,172.970,24.209,154.349
C02587=1071.518,28.518,434.989,172.971,24.212,154.350
C02588=1071.523,28.766,434.973,172.972,24.215,154.350
C02589=1071.529,29.016,434.958,172.974,24.217,154.350
C02590=1071.535,29.266,434.942,172.975,24.220,154.351
C02591=1071.541,29.515,434.926,172.976,24.222,154.351
C02592=1071.547,29.764,434.911,172.977,24.225,154.351
C02593=1071.552,30.014,434.896,172.979,24.228,154.352
C02594=1071.559,30.296,434.878,172.981,24.231,154.352
C02595=1071.566,30.579,434.861,172.982,24.234,154.353
C02596=1071.572,30.861,434.843,172.984,24.237,154.353
C02597=1071.578,31.143,434.826,172.986,24.240,154.353
C02598=1071.585,31.392,434.810,172.987,24.243,154.354
C02599=1071.591,31.642,434.794,172.988,24.245,154.354
C02600=1071.596,31.892,434.779,172.989,24.248,154.354
C02601=1071.603,32.140,434.763,172.991,24.250,154.355
C02602=1071.608,32.390,434.748,172.992,24.253,154.355
C02603=1071.614,32.640,434.732,172.993,24.256,154.355
C02604=1071.621,32.889,434.717,172.996,24.258,154.355
C02605=1071.626,33.139,434.700,172.997,24.261,154.356
C02606=1071.632,33.388,434.685,172.998,24.264,154.356
C02607=1071.638,33.637,434.670,173.000,24.266,154.356
C02608=1071.644,33.887,434.654,173.001,24.269,154.357
C02609=1071.650,34.136,434.638,173.002,24.271,154.357
C02610=1071.656,34.386,434.623,173.003,24.274,154.357
C02611=1071.662,34.635,434.607,173.005,24.277,154.358
C02612=1071.667,34.885,434.591,173.006,24.279,154.358
C02613=1071.673,35.134,434.575,173.007,24.281,154.358
C02614=1071.680,35.384,434.560,173.010,24.285,154.359
C02615=1071.685,35.633,434.544,173.011,24.287,154.359
C02616=1071.691,35.883,434.528,173.012,24.290,154.359
C02617=1071.698,36.132,434.513,173.013,24.292,154.360
C02618=1071.703,36.381,434.498,173.015,24.295,154.360
C02619=1071.709,36.631,434.481,173.016,24.298,154.360
C02620=1071.715,36.880,434.465,173.017,24.300,154.361
C02621=1071.721,37.130,434.450,173.019,24.302,154.361
C02622=1071.727,37.379,434.434,173.020,24.305,154.361
C02623=1071.733,37.629,434.418,173.021,24.308,154.362
C02624=1071.739,37.878,434.402,173.023,24.311,154.362
C02625=1071.745,38.127,434.386,173.025,24.313,154.362
C02626=1071.750,38.377,434.371,173.026,24.316,154.363
C02627=1071.756,38.626,434.355,173.027,24.319,154.363
C02628=1071.762,38.876,434.339,173.029,24.321,154.363
C02629=1071.768,39.125,434.323,173.030,24.324,154.364
C02630=1071.774,39.375,434.307,173.031,24.326,154.364
C02631=1071.780,39.625,434.291,173.033,24.329,154.364
C02632=1071.785,39.873,434.276,173.034,24.332,154.365
C02633=1071.791,40.123,434.259,173.035,24.335,154.365
C02634=1071.798,40.372,434.244,173.037,24.337,154.365
C02635=1071.803,40.622,434.228,173.039,24.340,154.366
C02636=1071.809,40.871,434.212,173.040,24.343,154.366
C02637=1071.815,41.120,434.196,173.041,24.345,154.366
C02638=1071.821,41.370,434.180,173.043,24.348,154.367
C02639=1071.827,41.620,434.164,173.044,24.350,154.367
C02640=1071.833,41.869,434.148,173.045,24.353,154.367
C02641=1071.838,42.118,434.132,173.047,24.356,154.368
C02642=1071.844,42.368,434.116,173.048,24.358,154.368
C02643=1071.850,42.617,434.100,173.049,24.361,154.368
C02644=1071.856,42.866,434.084,173.051,24.363,154.369
C02645=1071.861,43.116,434.067,173.053,24.367,154.369
C02646=1071.867,43.366,434.052,173.054,24.369,154.369
C02647=1071.873,43.615,434.036,173.055,24.372,154.370
C02648=1071.879,43.864,434.019,173.057,24.374,154.370
C02649=1071.885,44.114,434.003,173.058,24.377,154.370
C02650=1071.891,44.363,433.987,173.059,24.379,154.371
C02651=1071.897,44.613,433.971,173.060,24.382,154.371
C02652=1071.902,44.862,433.955,173.062,24.385,154.371
C02653=1071.908,45.111,433.939,173.063,24.388,154.372
C02654=1071.914,45.360,433.923,173.065,24.390,154.372
C02655=1071.920,45.610,433.907,173.067,24.393,154.372
C02656=1071.925,45.859,433.890,173.068,24.396,154.373
C02657=1071.931,46.109,433.873,173.069,24.399,154.373
C02658=1071.938,46.391,433.855,173.070,24.402,154.374
C02659=1071.944,46.673,433.837,173.072,24.405,154.374
C02660=1071.950,46.956,433.818,173.074,24.408,154.374
C02661=1071.957,47.238,433.800,173.075,24.411,154.375
C02662=1071.963,47.487,433.784,173.076,24.413,154.375
C02663=1071.969,47.736,433.768,173.078,24.416,154.375
C02664=1071.974,47.986,433.752,173.080,24.419,154.376
C02665=1071.980,48.236,433.736,173.081,24.422,154.376
C02666=1071.986,48.485,433.719,173.082,24.424,154.376
C02667=1071.991,48.735,433.703,173.084,24.427,154.377
C02668=1071.997,48.984,433.686,173.085,24.429,154.377
C02669=1072.003,49.233,433.670,173.086,24.432,154.377
C02670=1072.009,49.483,433.654,173.088,24.435,154.378
C02671=1072.015,49.732,433.637,173.089,24.437,154.378
C02672=1072.021,49.982,433.621,173.091,24.440,154.378
C02673=1072.026,50.231,433.605,173.092,24.443,154.379
C02674=1072.032,50.480,433.588,173.094,24.445,154.379
C02675=1072.038,50.730,433.572,173.095,24.448,154.379
C02676=1072.044,50.979,433.556,173.096,24.451,154.380
C02677=1072.050,51.229,433.539,173.098,24.454,154.380
C02678=1072.055,51.478,433.523,173.099,24.456,154.380
C02679=1072.061,51.728,433.506,173.100,24.459,154.381
C02680=1072.068,51.976,433.489,173.101,24.461,154.381
C02681=1072.073,52.226,433.473,173.104,24.464,154.381
C02682=1072.079,52.475,433.456,173.105,24.467,154.382
C02683=1072.085,52.725,433.440,173.106,24.469,154.382
C02684=1072.091,52.974,433.424,173.108,24.472,154.382
C02685=1072.097,53.223,433.408,173.109,24.475,154.383
C02686=1072.102,53.473,433.391,173.110,24.477,154.383
C02687=1072.108,53.722,433.374,173.112,24.480,154.383
C02688=1072.114,53.972,433.358,173.113,24.483,154.384
C02689=1072.120,54.221,433.342,173.115,24.485,154.384
C02690=1072.125,54.470,433.324,173.116,24.488,154.384
C02691=1072.131,54.719,433.308,173.118,24.491,154.385
C02692=1072.138,54.969,433.291,173.119,24.493,154.385
C02693=1072.144,55.219,433.275,173.120,24.496,154.385
C02694=1072.149,55.468,433.258,173.122,24.498,154.386
C02695=1072.155,55.718,433.242,173.123,24.501,154.386
C02696=1072.161,55.967,433.225,173.124,24.504,154.386
C02697=1072.167,56.216,433.209,173.126,24.507,154.387
C02698=1072.172,56.466,433.192,173.128,24.509,154.387
C02699=1072.178,56.715,433.176,173.129,24.512,154.387
C02700=1072.184,56.964,433.160,173.130,24.515,154.388
C02701=1072.190,57.213,433.143,173.132,24.517,154.388
C02702=1072.196,57.463,433.125,173.133,24.520,154.388
C02703=1072.202,57.713,433.109,173.134,24.522,154.389
C02704=1072.208,57.962,433.093,173.136,24.525,154.389
C02705=1072.214,58.211,433.075,173.138,24.528,154.389
C02706=1072.220,58.460,433.059,173.139,24.530,154.390
C02707=1072.226,58.710,433.043,173.141,24.533,154.390
C02708=1072.232,58.958,433.026,173.142,24.535,154.390
C02709=1072.238,59.209,433.009,173.143,24.538,154.391
C02710=1072.244,59.458,432.992,173.145,24.541,154.391
C02711=1072.250,59.708,432.976,173.146,24.543,154.391
C02712=1072.255,59.957,432.958,173.147,24.546,154.392
C02713=1072.261,60.206,432.942,173.150,24.549,154.392
C02714=1072.268,60.456,432.926,173.151,24.552,154.392
C02715=1072.274,60.705,432.909,173.152,24.554,154.393
C02716=1072.279,60.954,432.892,173.154,24.556,154.393
C02717=1072.285,61.204,432.876,173.155,24.559,154.393
C02718=1072.291,61.452,432.859,173.156,24.562,154.394
C02719=1072.297,61.703,432.841,173.157,24.564,154.394
C02720=1072.303,61.952,432.824,173.159,24.567,154.394
C02721=1072.309,62.201,432.808,173.161,24.570,154.395
C02722=1072.316,62.483,432.788,173.162,24.572,154.395
C02723=1072.323,62.766,432.770,173.164,24.575,154.395
C02724=1072.329,63.047,432.751,173.166,24.579,154.396
C02725=1072.336,63.329,432.732,173.167,24.582,154.396
C02726=1072.342,63.578,432.715,173.168,24.584,154.396
C02727=1072.348,63.828,432.697,173.171,24.587,154.397
C02728=1072.354,64.078,432.681,173.172,24.589,154.397
C02729=1072.360,64.326,432.664,173.173,24.592,154.397
C02730=1072.365,64.576,432.647,173.175,24.594,154.398
C02731=1072.372,64.825,432.630,173.176,24.597,154.398
C02732=1072.378,65.075,432.613,173.177,24.599,154.398
C02733=1072.384,65.324,432.596,173.178,24.602,154.399
C02734=1072.389,65.573,432.579,173.181,24.605,154.399
C02735=1072.395,65.822,432.562,173.182,24.608,154.399
C02736=1072.401,66.072,432.545,173.183,24.610,154.400
C02737=1072.407,66.322,432.528,173.185,24.613,154.400
C02738=1072.413,66.571,432.511,173.186,24.616,154.400
C02739=1072.418,66.820,432.494,173.187,24.618,154.401
C02740=1072.425,67.070,432.477,173.189,24.621,154.401
C02741=1072.430,67.319,432.460,173.191,24.624,154.401
C02742=1072.435,67.569,432.443,173.192,24.626,154.402
C02743=1072.442,67.817,432.426,173.194,24.629,154.402
C02744=1072.448,68.067,432.408,173.195,24.632,154.402
C02745=1072.454,68.316,432.392,173.196,24.634,154.403
C02746=1072.459,68.565,432.374,173.197,24.637,154.403
C02747=1072.464,68.815,432.357,173.199,24.639,154.403
C02748=1072.471,69.065,432.340,173.201,24.643,154.404
C02749=1072.477,69.314,432.322,173.202,24.645,154.404
C02750=1072.483,69.563,432.306,173.204,24.647,154.404
C02751=1072.488,69.812,432.288,173.205,24.650,154.405
C02752=1072.494,70.062,432.270,173.206,24.653,154.405
C02753=1072.500,70.311,432.254,173.208,24.655,154.406
C02754=1072.506,70.560,432.237,173.209,24.658,154.406
C02755=1072.511,70.809,432.219,173.211,24.661,154.406
C02756=1072.517,71.060,432.202,173.213,24.663,154.406
C02757=1072.523,71.308,432.185,173.214,24.666,154.407
C02758=1072.529,71.557,432.167,173.215,24.669,154.407
C02759=1072.535,71.808,432.150,173.217,24.672,154.408
C02760=1072.540,72.057,432.133,173.218,24.674,154.408
C02761=1072.547,72.305,432.116,173.219,24.677,154.408
C02762=1072.552,72.554,432.098,173.221,24.679,154.408
C02763=1072.558,72.805,432.081,173.223,24.682,154.409
C02764=1072.563,73.054,432.063,173.224,24.685,154.409
C02765=1072.570,73.303,432.046,173.225,24.688,154.410
C02766=1072.576,73.552,432.028,173.227,24.690,154.410
C02767=1072.581,73.802,432.011,173.228,24.692,154.410
C02768=1072.587,74.051,431.994,173.230,24.696,154.411
C02769=1072.593,74.300,431.977,173.232,24.698,154.411
C02770=1072.599,74.550,431.959,173.233,24.701,154.411
C02771=1072.604,74.799,431.941,173.234,24.703,154.412
C02772=1072.610,75.049,431.924,173.236,24.706,154.412
C02773=1072.616,75.298,431.907,173.237,24.708,154.412
C02774=1072.622,75.547,431.890,173.239,24.712,154.413
C02775=1072.628,75.796,431.872,173.241,24.714,154.413
C02776=1072.634,76.045,431.854,173.242,24.716,154.413
C02777=1072.639,76.295,431.837,173.243,24.719,154.414
C02778=1072.645,76.545,431.819,173.245,24.722,154.414
C02779=1072.651,76.794,431.802,173.246,24.724,154.414
C02780=1072.657,77.043,431.785,173.248,24.727,154.414
C02781=1072.663,77.292,431.767,173.249,24.730,154.415
C02782=1072.668,77.541,431.749,173.251,24.732,154.415
C02783=1072.674,77.791,431.731,173.252,24.735,154.415
C02784=1072.680,78.040,431.714,173.253,24.738,154.416
C02785=1072.686,78.289,431.696,173.255,24.740,154.416
C02786=1072.692,78.571,431.677,173.257,24.743,154.417
C02787=1072.699,78.854,431.657,173.258,24.746,154.417
C02788=1072.705,79.135,431.637,173.260,24.749,154.417
C02789=1072.712,79.418,431.617,173.262,24.752,154.418
C02790=1072.717,79.667,431.599,173.263,24.755,154.418
C02791=1072.724,79.916,431.581,173.265,24.758,154.418
C02792=1072.729,80.165,431.564,173.267,24.761,154.419
C02793=1072.735,80.414,431.546,173.268,24.763,154.419
C02794=1072.741,80.664,431.528,173.269,24.766,154.419
C02795=1072.746,80.913,431.511,173.271,24.768,154.420
C02796=1072.752,81.162,431.493,173.272,24.771,154.420
C02797=1072.758,81.412,431.475,173.274,24.774,154.420
C02798=1072.763,81.661,431.458,173.276,24.776,154.421
C02799=1072.770,81.911,431.440,173.277,24.779,154.421
C02800=1072.775,82.160,431.422,173.278,24.782,154.421
C02801=1072.781,82.409,431.405,173.279,24.784,154.422
C02802=1072.787,82.659,431.387,173.281,24.787,154.422
C02803=1072.793,82.907,431.368,173.283,24.790,154.422
C02804=1072.799,83.157,431.350,173.284,24.792,154.423
C02805=1072.804,83.406,431.333,173.286,24.795,154.423
C02806=1072.810,83.655,431.315,173.287,24.798,154.423
C02807=1072.816,83.905,431.297,173.288,24.800,154.424
C02808=1072.821,84.154,431.280,173.291,24.803,154.424
C02809=1072.827,84.403,431.262,173.292,24.806,154.425
C02810=1072.832,84.653,431.244,173.293,24.808,154.425
C02811=1072.838,84.902,431.226,173.295,24.811,154.425
C02812=1072.844,85.151,431.207,173.296,24.814,154.426
C02813=1072.850,85.401,431.190,173.297,24.816,154.426
C02814=1072.856,85.650,431.172,173.300,24.819,154.426
C02815=1072.862,85.899,431.154,173.301,24.822,154.426
C02816=1072.867,86.148,431.136,173.302,24.824,154.427
C02817=1072.874,86.398,431.118,173.304,24.827,154.427
C02818=1072.879,86.647,431.100,173.305,24.829,154.427
C02819=1072.885,86.896,431.082,173.307,24.832,154.428
C02820=1072.891,87.145,431.065,173.309,24.835,154.428
C02821=1072.897,87.395,431.047,173.310,24.838,154.429
C02822=1072.902,87.644,431.028,173.311,24.840,154.429
C02823=1072.908,87.894,431.010,173.313,24.842,154.429
C02824=1072.914,88.143,430.992,173.315,24.845,154.429
C02825=1072.920,88.392,430.974,173.316,24.848,154.430
C02826=1072.926,88.604,430.959,173.318,24.850,154.430
C02827=1072.930,88.816,430.944,173.319,24.852,154.430
C02828=1072.935,89.029,430.929,173.320,24.854,154.431
C02829=1072.940,89.241,430.912,173.321,24.857,154.431
C02830=1072.946,89.454,430.897,173.322,24.859,154.431
C02831=1072.950,89.666,430.882,173.324,24.861,154.431
C02832=1072.955,89.878,430.867,173.325,24.863,154.432
C02833=1072.960,90.091,430.851,173.327,24.866,154.432
C02834=1072.966,90.340,430.834,173.328,24.868,154.432
C02835=1072.972,90.589,430.816,173.329,24.871,154.433
C02836=1072.978,90.838,430.797,173.331,24.873,154.433
C02837=1072.983,91.088,430.779,173.333,24.876,154.433
C02838=1072.989,91.337,430.760,173.334,24.879,154.434
C02839=1072.995,91.586,430.743,173.336,24.882,154.434
C02840=1073.000,91.836,430.724,173.337,24.884,154.434
C02841=1073.006,92.084,430.706,173.338,24.887,154.435
C02842=1073.012,92.334,430.688,173.341,24.890,154.435
C02843=1073.017,92.584,430.670,173.342,24.892,154.435
C02844=1073.023,92.833,430.651,173.343,24.895,154.436
C02845=1073.029,93.082,430.633,173.345,24.897,154.436
C02846=1073.035,93.331,430.614,173.346,24.900,154.436
C02847=1073.040,93.580,430.597,173.348,24.903,154.437
C02848=1073.047,93.829,430.578,173.350,24.905,154.437
C02849=1073.052,94.079,430.559,173.351,24.908,154.437
C02850=1073.060,94.435,430.533,173.353,24.912,154.438
C02851=1073.068,94.791,430.507,173.355,24.915,154.438
C02852=1073.077,95.146,430.481,173.358,24.920,154.439
C02853=1073.085,95.502,430.455,173.360,24.923,154.439
C02854=1073.090,95.751,430.436,173.362,24.926,154.440
C02855=1073.096,96.001,430.418,173.363,24.928,154.440
C02856=1073.103,96.250,430.400,173.364,24.931,154.440
C02857=1073.107,96.499,430.381,173.367,24.933,154.440
C02858=1073.114,96.748,430.363,173.368,24.936,154.441
C02859=1073.119,96.998,430.345,173.369,24.939,154.441
C02860=1073.125,97.247,430.326,173.371,24.942,154.442
C02861=1073.131,97.497,430.308,173.373,24.944,154.442
C02862=1073.136,97.745,430.289,173.374,24.947,154.442
C02863=1073.143,97.995,430.270,173.376,24.949,154.443
C02864=1073.148,98.245,430.252,173.377,24.952,154.443
C02865=1073.154,98.493,430.234,173.378,24.954,154.443
C02866=1073.160,98.743,430.216,173.381,24.957,154.443
C02867=1073.166,98.992,430.196,173.382,24.960,154.444
C02868=1073.172,99.241,430.178,173.383,24.963,154.444
C02869=1073.177,99.491,430.160,173.385,24.965,154.444
C02870=1073.183,99.740,430.141,173.387,24.968,154.445
C02871=1073.188,99.989,430.122,173.388,24.970,154.445
C02872=1073.195,100.238,430.104,173.390,24.973,154.445
C02873=1073.201,100.487,430.086,173.391,24.975,154.446
C02874=1073.206,100.736,430.067,173.393,24.978,154.446
C02875=1073.212,100.986,430.049,173.395,24.981,154.446
C02876=1073.218,101.235,430.029,173.396,24.983,154.447
C02877=1073.224,101.484,430.011,173.397,24.986,154.447
C02878=1073.229,101.734,429.993,173.400,24.989,154.447
C02879=1073.235,101.983,429.973,173.401,24.991,154.448
C02880=1073.241,102.232,429.955,173.402,24.994,154.448
C02881=1073.246,102.481,429.936,173.404,24.997,154.448
C02882=1073.252,102.731,429.917,173.405,24.999,154.449
C02883=1073.257,102.980,429.899,173.407,25.002,154.449
C02884=1073.263,103.229,429.880,173.409,25.004,154.449
C02885=1073.270,103.478,429.861,173.410,25.007,154.450
C02886=1073.275,103.727,429.842,173.411,25.010,154.450
C02887=1073.280,103.977,429.824,173.414,25.012,154.450
C02888=1073.286,104.226,429.805,173.415,25.015,154.451
C02889=1073.292,104.475,429.786,173.416,25.018,154.451
C02890=1073.297,104.724,429.767,173.418,25.020,154.451
C02891=1073.304,104.973,429.748,173.420,25.023,154.452
C02892=1073.309,105.223,429.729,173.421,25.025,154.452
C02893=1073.314,105.472,429.711,173.423,25.028,154.452
C02894=1073.321,105.721,429.692,173.424,25.031,154.453
C02895=1073.326,105.971,429.673,173.426,25.033,154.453
C02896=1073.332,106.220,429.654,173.428,25.036,154.453
C02897=1073.338,106.468,429.636,173.429,25.038,154.454
C02898=1073.343,106.718,429.616,173.432,25.041,154.454
C02899=1073.349,106.967,429.597,173.433,25.044,154.454
C02900=1073.356,107.216,429.578,173.434,25.046,154.455
C02901=1073.361,107.465,429.560,173.436,25.049,154.455
C02902=1073.366,107.715,429.540,173.438,25.052,154.455
C02903=1073.372,107.965,429.522,173.439,25.054,154.455
C02904=1073.378,108.214,429.503,173.441,25.057,154.456
C02905=1073.384,108.463,429.484,173.442,25.059,154.456
C02906=1073.389,108.712,429.465,173.444,25.062,154.456
C02907=1073.395,108.961,429.446,173.446,25.064,154.457
C02908=1073.401,109.211,429.427,173.447,25.067,154.457
C02909=1073.407,109.460,429.408,173.448,25.070,154.457
C02910=1073.413,109.709,429.389,173.451,25.072,154.458
C02911=1073.418,109.958,429.370,173.452,25.075,154.458
C02912=1073.424,110.207,429.351,173.453,25.077,154.458
C02913=1073.430,110.457,429.332,173.456,25.080,154.459
C02914=1073.437,110.739,429.310,173.457,25.083,154.459
C02915=1073.443,111.021,429.289,173.459,25.086,154.459
C02916=1073.450,111.303,429.267,173.461,25.089,154.460
C02917=1073.456,111.584,429.246,173.463,25.092,154.460
C02918=1073.461,111.834,429.226,173.464,25.095,154.460
C02919=1073.468,112.083,429.208,173.466,25.097,154.461
C02920=1073.474,112.332,429.188,173.468,25.100,154.461
C02921=1073.480,112.581,429.169,173.469,25.102,154.461
C02922=1073.485,112.830,429.150,173.471,25.105,154.462
C02923=1073.490,113.079,429.130,173.473,25.108,154.462
C02924=1073.496,113.329,429.111,173.474,25.110,154.462
C02925=1073.502,113.578,429.092,173.476,25.113,154.463
C02926=1073.508,113.827,429.073,173.477,25.115,154.463
C02927=1073.514,114.076,429.053,173.479,25.118,154.463
C02928=1073.520,114.326,429.034,173.481,25.120,154.464
C02929=1073.525,114.574,429.015,173.482,25.123,154.464
C02930=1073.531,114.824,428.996,173.484,25.126,154.464
C02931=1073.536,115.073,428.977,173.486,25.129,154.465
C02932=1073.542,115.323,428.958,173.487,25.131,154.465
C02933=1073.548,115.572,428.938,173.489,25.133,154.465
C02934=1073.552,115.821,428.918,173.491,25.137,154.466
C02935=1073.558,116.070,428.899,173.492,25.139,154.466
C02936=1073.564,116.319,428.880,173.494,25.142,154.466
C02937=1073.570,116.568,428.860,173.496,25.145,154.467
C02938=1073.575,116.818,428.840,173.497,25.147,154.467
C02939=1073.581,117.067,428.821,173.499,25.150,154.467
C02940=1073.586,117.316,428.802,173.501,25.152,154.468
C02941=1073.592,117.565,428.782,173.502,25.155,154.468
C02942=1073.598,117.814,428.763,173.504,25.158,154.468
C02943=1073.604,118.064,428.744,173.505,25.160,154.469
C02944=1073.610,118.312,428.724,173.507,25.163,154.469
C02945=1073.615,118.562,428.705,173.509,25.165,154.469
C02946=1073.620,118.812,428.685,173.510,25.168,154.470
C02947=1073.626,119.060,428.665,173.512,25.171,154.470
C02948=1073.631,119.309,428.646,173.514,25.173,154.470
C02949=1073.637,119.558,428.627,173.515,25.176,154.471
C02950=1073.643,119.807,428.607,173.517,25.179,154.471
C02951=1073.649,120.057,428.588,173.519,25.182,154.471
C02952=1073.654,120.306,428.568,173.520,25.184,154.472
C02953=1073.660,120.555,428.548,173.522,25.187,154.472
C02954=1073.666,120.804,428.529,173.524,25.189,154.472
C02955=1073.671,121.054,428.509,173.525,25.192,154.472
C02956=1073.677,121.303,428.489,173.528,25.194,154.473
C02957=1073.683,121.552,428.469,173.529,25.197,154.473
C02958=1073.689,121.801,428.450,173.530,25.200,154.473
C02959=1073.694,122.051,428.431,173.532,25.202,154.474
C02960=1073.700,122.299,428.411,173.534,25.205,154.474
C02961=1073.705,122.548,428.392,173.535,25.207,154.474
C02962=1073.711,122.797,428.371,173.537,25.210,154.475
C02963=1073.716,123.047,428.352,173.539,25.213,154.475
C02964=1073.722,123.296,428.332,173.540,25.215,154.475
C02965=1073.728,123.545,428.313,173.542,25.217,154.476
C02966=1073.734,123.794,428.293,173.544,25.221,154.476
C02967=1073.740,124.043,428.274,173.546,25.223,154.476
C02968=1073.745,124.292,428.253,173.547,25.225,154.477
C02969=1073.751,124.542,428.234,173.549,25.228,154.477
C02970=1073.757,124.791,428.214,173.551,25.231,154.477
C02971=1073.763,125.039,428.194,173.552,25.233,154.478
C02972=1073.768,125.289,428.175,173.554,25.236,154.478
C02973=1073.774,125.538,428.155,173.556,25.239,154.478
C02974=1073.779,125.787,428.135,173.557,25.241,154.479
C02975=1073.785,126.036,428.115,173.559,25.244,154.479
C02976=1073.791,126.286,428.096,173.561,25.246,154.479
C02977=1073.798,126.535,428.076,173.563,25.249,154.479
C02978=1073.803,126.817,428.053,173.565,25.251,154.480
C02979=1073.810,127.099,428.031,173.567,25.255,154.480
C02980=1073.816,127.381,428.008,173.569,25.258,154.480
C02981=1073.824,127.662,427.986,173.570,25.260,154.481
C02982=1073.829,127.912,427.966,173.573,25.263,154.481
C02983=1073.835,128.161,427.946,173.574,25.266,154.481
C02984=1073.841,128.410,427.926,173.576,25.268,154.482
C02985=1073.846,128.659,427.907,173.578,25.271,154.482
C02986=1073.852,128.908,427.886,173.579,25.273,154.482
C02987=1073.858,129.157,427.866,173.581,25.276,154.483
C02988=1073.864,129.407,427.847,173.583,25.278,154.483
C02989=1073.870,129.656,427.827,173.584,25.281,154.483
C02990=1073.876,129.905,427.807,173.586,25.283,154.484
C02991=1073.881,130.154,427.786,173.588,25.286,154.484
C02992=1073.887,130.404,427.767,173.590,25.288,154.484
C02993=1073.893,130.652,427.747,173.592,25.291,154.484
C02994=1073.899,130.901,427.727,173.593,25.293,154.485
C02995=1073.904,131.150,427.706,173.595,25.296,154.485
C02996=1073.910,131.400,427.687,173.597,25.299,154.485
C02997=1073.916,131.649,427.667,173.598,25.301,154.486
C02998=1073.922,131.898,427.647,173.600,25.304,154.486
C02999=1073.928,132.147,427.626,173.602,25.306,154.486
C03000=1073.934,132.396,427.606,173.604,25.309,154.487
C03001=1073.939,132.646,427.586,173.606,25.312,154.487
C03002=1073.945,132.895,427.567,173.607,25.314,154.487
C03003=1073.950,133.144,427.546,173.609,25.316,154.487
C03004=1073.956,133.392,427.526,173.611,25.319,154.488
C03005=1073.962,133.642,427.505,173.612,25.322,154.488
C03006=1073.968,133.891,427.485,173.614,25.324,154.488
C03007=1073.973,134.140,427.465,173.616,25.327,154.489
C03008=1073.979,134.389,427.445,173.618,25.330,154.489
C03009=1073.984,134.639,427.425,173.620,25.332,154.489
C03010=1073.990,134.888,427.405,173.621,25.334,154.490
C03011=1073.995,135.137,427.384,173.623,25.337,154.490
C03012=1074.001,135.386,427.364,173.625,25.340,154.490
C03013=1074.007,135.635,427.343,173.626,25.342,154.491
C03014=1074.013,135.884,427.323,173.629,25.345,154.491
C03015=1074.018,136.133,427.303,173.630,25.348,154.491
C03016=1074.024,136.382,427.283,173.632,25.350,154.492
C03017=1074.029,136.631,427.262,173.634,25.353,154.492
C03018=1074.035,136.880,427.242,173.635,25.356,154.492
C03019=1074.041,137.130,427.221,173.638,25.358,154.492
C03020=1074.047,137.379,427.202,173.639,25.360,154.493
C03021=1074.053,137.628,427.181,173.641,25.363,154.493
C03022=1074.059,137.877,427.161,173.643,25.366,154.493
C03023=1074.064,138.126,427.140,173.644,25.368,154.494
C03024=1074.070,138.376,427.120,173.647,25.371,154.494
C03025=1074.076,138.624,427.100,173.648,25.373,154.494
C03026=1074.081,138.874,427.079,173.649,25.376,154.495
C03027=1074.087,139.122,427.059,173.652,25.379,154.495
C03028=1074.092,139.371,427.038,173.653,25.381,154.495
C03029=1074.098,139.621,427.017,173.655,25.384,154.495
C03030=1074.104,139.869,426.997,173.657,25.386,154.496
C03031=1074.110,140.119,426.976,173.659,25.389,154.496
C03032=1074.116,140.367,426.956,173.661,25.391,154.496
C03033=1074.121,140.617,426.935,173.662,25.394,154.497
C03034=1074.127,140.866,426.915,173.664,25.397,154.497
C03035=1074.132,141.115,426.894,173.666,25.399,154.497
C03036=1074.138,141.364,426.874,173.668,25.402,154.498
C03037=1074.143,141.613,426.853,173.670,25.404,154.498
C03038=1074.149,141.863,426.832,173.671,25.407,154.498
C03039=1074.155,142.112,426.812,173.673,25.410,154.499
C03040=1074.161,142.361,426.792,173.675,25.412,154.499
C03041=1074.166,142.609,426.770,173.677,25.415,154.499
C03042=1074.172,142.891,426.748,173.679,25.418,154.500
C03043=1074.179,143.173,426.724,173.681,25.421,154.500
C03044=1074.185,143.455,426.700,173.683,25.424,154.500
C03045=1074.191,143.737,426.677,173.685,25.426,154.501
C03046=1074.197,143.987,426.656,173.687,25.429,154.501
C03047=1074.203,144.235,426.636,173.689,25.432,154.501
C03048=1074.209,144.484,426.615,173.690,25.434,154.502
C03049=1074.215,144.734,426.594,173.693,25.437,154.502
C03050=1074.220,144.983,426.573,173.694,25.440,154.502
C03051=1074.226,145.231,426.553,173.695,25.442,154.503
C03052=1074.231,145.480,426.532,173.698,25.444,154.503
C03053=1074.237,145.730,426.511,173.699,25.447,154.503
C03054=1074.243,145.978,426.490,173.702,25.449,154.503
C03055=1074.248,146.228,426.469,173.703,25.452,154.504
C03056=1074.255,146.477,426.449,173.705,25.455,154.504
C03057=1074.260,146.726,426.428,173.707,25.457,154.504
C03058=1074.266,146.975,426.407,173.709,25.460,154.505
C03059=1074.271,147.225,426.386,173.711,25.462,154.505
C03060=1074.277,147.473,426.365,173.713,25.465,154.505
C03061=1074.283,147.722,426.345,173.714,25.468,154.505
C03062=1074.289,147.971,426.323,173.717,25.470,154.506
C03063=1074.294,148.220,426.303,173.718,25.472,154.506
C03064=1074.300,148.469,426.282,173.719,25.475,154.506
C03065=1074.306,148.719,426.261,173.722,25.478,154.507
C03066=1074.311,148.968,426.240,173.723,25.480,154.507
C03067=1074.317,149.216,426.219,173.726,25.483,154.507
C03068=1074.322,149.466,426.198,173.727,25.486,154.508
C03069=1074.328,149.715,426.177,173.729,25.488,154.508
C03070=1074.334,149.964,426.156,173.731,25.491,154.508
C03071=1074.339,150.213,426.135,173.733,25.493,154.508
C03072=1074.345,150.462,426.114,173.735,25.496,154.509
C03073=1074.351,150.711,426.092,173.737,25.499,154.509
C03074=1074.356,150.960,426.072,173.738,25.501,154.509
C03075=1074.362,151.209,426.051,173.741,25.504,154.510
C03076=1074.368,151.459,426.030,173.742,25.506,154.510
C03077=1074.373,151.707,426.008,173.744,25.509,154.510
C03078=1074.379,151.956,425.987,173.746,25.511,154.511
C03079=1074.385,152.205,425.966,173.748,25.514,154.511
C03080=1074.390,152.454,425.945,173.750,25.517,154.511
C03081=1074.396,152.704,425.924,173.752,25.519,154.512
C03082=1074.401,152.952,425.903,173.753,25.522,154.512
C03083=1074.407,153.201,425.881,173.756,25.524,154.512
C03084=1074.413,153.451,425.860,173.757,25.527,154.512
C03085=1074.418,153.699,425.839,173.760,25.530,154.513
C03086=1074.425,153.948,425.818,173.761,25.532,154.513
C03087=1074.430,154.197,425.797,173.763,25.535,154.513
C03088=1074.436,154.447,425.775,173.765,25.537,154.514
C03089=1074.442,154.695,425.754,173.767,25.540,154.514
C03090=1074.447,154.944,425.734,173.769,25.542,154.514
C03091=1074.453,155.193,425.712,173.771,25.545,154.515
C03092=1074.459,155.442,425.691,173.772,25.547,154.515
C03093=1074.464,155.692,425.670,173.775,25.550,154.515
C03094=1074.469,155.941,425.648,173.776,25.553,154.516
C03095=1074.475,156.190,425.626,173.778,25.555,154.516
C03096=1074.481,156.438,425.605,173.780,25.558,154.516
C03097=1074.487,156.688,425.584,173.782,25.560,154.516
C03098=1074.492,156.937,425.563,173.784,25.563,154.517
C03099=1074.498,157.185,425.542,173.786,25.566,154.517
C03100=1074.503,157.435,425.519,173.787,25.568,154.517
C03101=1074.509,157.684,425.499,173.790,25.571,154.518
C03102=1074.515,157.933,425.477,173.791,25.573,154.518
C03103=1074.520,158.182,425.456,173.794,25.576,154.518
C03104=1074.527,158.431,425.434,173.795,25.578,154.519
C03105=1074.531,158.680,425.412,173.797,25.581,154.519
C03106=1074.539,158.962,425.389,173.800,25.584,154.519
C03107=1074.545,159.243,425.364,173.802,25.587,154.520
C03108=1074.552,159.524,425.340,173.804,25.590,154.520
C03109=1074.557,159.806,425.316,173.806,25.593,154.520
C03110=1074.564,160.056,425.294,173.808,25.595,154.520
C03111=1074.568,160.304,425.272,173.810,25.598,154.521
C03112=1074.575,160.554,425.251,173.812,25.600,154.521
C03113=1074.580,160.802,425.229,173.814,25.603,154.521
C03114=1074.586,161.051,425.208,173.816,25.606,154.522
C03115=1074.592,161.300,425.186,173.818,25.608,154.522
C03116=1074.597,161.549,425.164,173.819,25.611,154.522
C03117=1074.603,161.798,425.143,173.822,25.614,154.523
C03118=1074.608,162.047,425.121,173.823,25.616,154.523
C03119=1074.614,162.296,425.099,173.826,25.619,154.523
C03120=1074.619,162.545,425.077,173.828,25.622,154.524
C03121=1074.625,162.794,425.056,173.829,25.624,154.524
C03122=1074.630,163.043,425.034,173.831,25.627,154.524
C03123=1074.636,163.292,425.012,173.833,25.630,154.525
C03124=1074.641,163.541,424.990,173.835,25.632,154.525
C03125=1074.646,163.790,424.968,173.837,25.635,154.525
C03126=1074.652,164.039,424.947,173.839,25.638,154.525
C03127=1074.657,164.288,424.925,173.841,25.640,154.526
C03128=1074.663,164.537,424.903,173.843,25.643,154.526
C03129=1074.668,164.786,424.881,173.845,25.646,154.526
C03130=1074.674,165.035,424.860,173.847,25.648,154.527
C03131=1074.679,165.284,424.838,173.849,25.651,154.527
C03132=1074.685,165.533,424.816,173.850,25.653,154.527
C03133=1074.690,165.782,424.794,173.853,25.656,154.528
C03134=1074.696,166.031,424.772,173.855,25.659,154.528
C03135=1074.701,166.280,424.750,173.856,25.661,154.528
C03136=1074.707,166.529,424.728,173.859,25.664,154.529
C03137=1074.713,166.778,424.706,173.860,25.667,154.529
C03138=1074.718,167.027,424.684,173.863,25.669,154.529
C03139=1074.724,167.276,424.662,173.864,25.672,154.530
C03140=1074.729,167.525,424.640,173.866,25.675,154.530
C03141=1074.734,167.774,424.618,173.869,25.677,154.530
C03142=1074.740,168.023,424.597,173.870,25.680,154.530
C03143=1074.746,168.272,424.574,173.873,25.682,154.531
C03144=1074.752,168.521,424.552,173.874,25.685,154.531
C03145=1074.757,168.770,424.530,173.876,25.688,154.531
C03146=1074.762,169.019,424.508,173.879,25.690,154.532
C03147=1074.769,169.268,424.486,173.880,25.693,154.532
C03148=1074.773,169.517,424.464,173.882,25.696,154.532
C03149=1074.780,169.766,424.442,173.884,25.698,154.533
C03150=1074.784,170.015,424.420,173.886,25.701,154.533
C03151=1074.790,170.263,424.397,173.889,25.704,154.533
C03152=1074.796,170.513,424.376,173.890,25.706,154.534
C03153=1074.801,170.761,424.354,173.892,25.709,154.534
C03154=1074.808,171.010,424.332,173.895,25.712,154.534
C03155=1074.813,171.260,424.309,173.896,25.714,154.535
C03156=1074.818,171.508,424.287,173.899,25.717,154.535
C03157=1074.824,171.757,424.265,173.900,25.719,154.535
C03158=1074.830,172.006,424.243,173.902,25.722,154.535
C03159=1074.835,172.255,424.220,173.905,25.725,154.536
C03160=1074.841,172.504,424.199,173.906,25.727,154.536
C03161=1074.846,172.753,424.176,173.909,25.730,154.536
C03162=1074.852,173.002,424.153,173.911,25.733,154.537
C03163=1074.858,173.251,424.132,173.912,25.735,154.537
C03164=1074.863,173.500,424.109,173.915,25.738,154.537
C03165=1074.869,173.749,424.087,173.917,25.740,154.537
C03166=1074.875,173.997,424.065,173.918,25.743,154.538
C03167=1074.880,174.247,424.043,173.921,25.746,154.538
C03168=1074.886,174.495,424.020,173.922,25.748,154.538
C03169=1074.892,174.745,423.998,173.925,25.750,154.539
C03170=1074.898,175.025,423.973,173.927,25.754,154.539
C03171=1074.905,175.307,423.948,173.929,25.757,154.539
C03172=1074.910,175.588,423.922,173.932,25.759,154.540
C03173=1074.917,175.870,423.897,173.934,25.762,154.540
C03174=1074.924,176.119,423.875,173.936,25.765,154.540
C03175=1074.928,176.367,423.853,173.938,25.767,154.541
C03176=1074.934,176.616,423.830,173.940,25.770,154.541
C03177=1074.940,176.865,423.808,173.942,25.773,154.541
C03178=1074.946,177.114,423.785,173.944,25.775,154.542
C03179=1074.952,177.363,423.762,173.946,25.778,154.542
C03180=1074.957,177.612,423.740,173.949,25.781,154.542
C03181=1074.963,177.861,423.718,173.950,25.783,154.542
C03182=1074.969,178.110,423.695,173.952,25.786,154.543
C03183=1074.974,178.359,423.673,173.955,25.789,154.543
C03184=1074.980,178.608,423.650,173.956,25.791,154.543
C03185=1074.986,178.857,423.628,173.959,25.793,154.544
C03186=1074.991,179.105,423.606,173.961,25.796,154.544
C03187=1074.997,179.354,423.583,173.963,25.799,154.544
C03188=1075.003,179.603,423.560,173.965,25.801,154.545
C03189=1075.009,179.852,423.538,173.967,25.804,154.545
C03190=1075.015,180.101,423.515,173.970,25.807,154.545
C03191=1075.020,180.350,423.492,173.971,25.809,154.545
C03192=1075.026,180.600,423.470,173.974,25.811,154.546
C03193=1075.032,180.848,423.448,173.976,25.815,154.546
C03194=1075.037,181.096,423.425,173.977,25.817,154.546
C03195=1075.043,181.345,423.402,173.980,25.819,154.547
C03196=1075.048,181.595,423.380,173.982,25.822,154.547
C03197=1075.055,181.843,423.358,173.985,25.825,154.547
C03198=1075.061,182.092,423.335,173.986,25.827,154.547
C03199=1075.066,182.341,423.312,173.988,25.830,154.548
C03200=1075.072,182.590,423.289,173.991,25.833,154.548
C03201=1075.078,182.840,423.267,173.992,25.835,154.548
C03202=1075.084,183.088,423.244,173.995,25.837,154.549
C03203=1075.090,183.337,423.221,173.997,25.840,154.549
C03204=1075.095,183.586,423.198,173.999,25.843,154.549
C03205=1075.101,183.835,423.175,174.001,25.845,154.549
C03206=1075.107,184.084,423.152,174.003,25.848,154.550
C03207=1075.113,184.332,423.130,174.006,25.851,154.550
C03208=1075.119,184.581,423.107,174.007,25.853,154.550
C03209=1075.125,184.831,423.085,174.009,25.856,154.551
C03210=1075.130,185.080,423.062,174.012,25.858,154.551
C03211=1075.135,185.328,423.039,174.014,25.861,154.551
C03212=1075.140,185.577,423.016,174.016,25.863,154.552
C03213=1075.146,185.826,422.993,174.018,25.867,154.552
C03214=1075.152,186.075,422.970,174.020,25.869,154.552
C03215=1075.158,186.324,422.947,174.023,25.872,154.552
C03216=1075.163,186.573,422.924,174.024,25.875,154.553
C03217=1075.168,186.822,422.901,174.027,25.877,154.553
C03218=1075.174,187.071,422.878,174.029,25.880,154.553
C03219=1075.180,187.320,422.855,174.031,25.883,154.554
C03220=1075.185,187.568,422.832,174.033,25.885,154.554
C03221=1075.190,187.817,422.809,174.035,25.888,154.554
C03222=1075.196,188.066,422.786,174.037,25.891,154.555
C03223=1075.202,188.314,422.762,174.040,25.893,154.555
C03224=1075.207,188.563,422.739,174.041,25.896,154.555
C03225=1075.212,188.812,422.715,174.044,25.899,154.556
C03226=1075.218,189.061,422.693,174.046,25.902,154.556
C03227=1075.224,189.310,422.670,174.048,25.905,154.556
C03228=1075.230,189.559,422.647,174.050,25.907,154.557
C03229=1075.235,189.808,422.623,174.052,25.910,154.557
C03230=1075.240,190.057,422.600,174.054,25.913,154.557
C03231=1075.246,190.305,422.576,174.057,25.915,154.558
C03232=1075.251,190.555,422.553,174.058,25.918,154.558
C03233=1075.257,190.804,422.530,174.061,25.920,154.558
C03234=1075.263,191.084,422.505,174.063,25.924,154.559
C03235=1075.269,191.365,422.478,174.065,25.927,154.559
C03236=1075.276,191.647,422.451,174.069,25.930,154.559
C03237=1075.283,191.927,422.425,174.071,25.933,154.560
C03238=1075.288,192.176,422.402,174.073,25.936,154.560
C03239=1075.293,192.425,422.379,174.075,25.938,154.560
C03240=1075.299,192.673,422.355,174.077,25.941,154.561
C03241=1075.304,192.922,422.332,174.079,25.944,154.561
C03242=1075.310,193.171,422.309,174.082,25.946,154.561
C03243=1075.316,193.420,422.286,174.084,25.949,154.561
C03244=1075.321,193.669,422.262,174.086,25.952,154.562
C03245=1075.327,193.918,422.239,174.088,25.954,154.562
C03246=1075.333,194.166,422.216,174.090,25.957,154.562
C03247=1075.338,194.415,422.191,174.093,25.960,154.563
C03248=1075.344,194.664,422.168,174.095,25.963,154.563
C03249=1075.350,194.914,422.145,174.097,25.965,154.563
C03250=1075.355,195.162,422.121,174.099,25.968,154.564
C03251=1075.361,195.411,422.098,174.101,25.971,154.564
C03252=1075.367,195.659,422.074,174.104,25.973,154.564
C03253=1075.372,195.908,422.051,174.106,25.976,154.565
C03254=1075.378,196.157,422.028,174.107,25.979,154.565
C03255=1075.384,196.406,422.004,174.110,25.981,154.565
C03256=1075.389,196.655,421.981,174.112,25.984,154.566
C03257=1075.395,196.903,421.957,174.115,25.987,154.566
C03258=1075.401,197.153,421.934,174.117,25.989,154.566
C03259=1075.406,197.401,421.909,174.119,25.992,154.567
C03260=1075.412,197.650,421.886,174.121,25.995,154.567
C03261=1075.417,197.899,421.862,174.123,25.997,154.567
C03262=1075.423,198.148,421.839,174.125,26.000,154.567
C03263=1075.429,198.396,421.816,174.128,26.003,154.568
C03264=1075.435,198.646,421.792,174.130,26.006,154.568
C03265=1075.441,198.894,421.768,174.133,26.009,154.568
C03266=1075.446,199.143,421.744,174.135,26.011,154.569
C03267=1075.452,199.392,421.721,174.137,26.013,154.569
C03268=1075.458,199.641,421.698,174.139,26.017,154.569
C03269=1075.463,199.890,421.673,174.141,26.019,154.570
C03270=1075.469,200.138,421.650,174.144,26.022,154.570
C03271=1075.474,200.387,421.626,174.146,26.025,154.570
C03272=1075.481,200.636,421.602,174.148,26.027,154.571
C03273=1075.486,200.884,421.579,174.151,26.030,154.571
C03274=1075.492,201.134,421.555,174.152,26.033,154.571
C03275=1075.498,201.382,421.531,174.155,26.035,154.571
C03276=1075.503,201.631,421.508,174.157,26.038,154.572
C03277=1075.509,201.880,421.484,174.159,26.040,154.572
C03278=1075.515,202.129,421.459,174.162,26.044,154.572
C03279=1075.521,202.378,421.436,174.164,26.046,154.573
C03280=1075.526,202.626,421.412,174.167,26.049,154.573
C03281=1075.532,202.875,421.388,174.169,26.052,154.573
C03282=1075.538,203.124,421.364,174.171,26.054,154.574
C03283=1075.543,203.373,421.340,174.173,26.057,154.574
C03284=1075.549,203.621,421.317,174.175,26.060,154.574
C03285=1075.554,203.870,421.292,174.177,26.063,154.575
C03286=1075.560,204.119,421.268,174.180,26.065,154.575
C03287=1075.566,204.368,421.245,174.182,26.069,154.575
C03288=1075.571,204.617,421.220,174.185,26.071,154.576
C03289=1075.577,204.865,421.196,174.187,26.074,154.576
C03290=1075.582,205.114,421.172,174.189,26.077,154.576
C03291=1075.589,205.363,421.148,174.192,26.080,154.577
C03292=1075.594,205.611,421.124,174.193,26.082,154.577
C03293=1075.599,205.861,421.100,174.196,26.085,154.577
C03294=1075.605,206.109,421.077,174.198,26.088,154.578
C03295=1075.611,206.358,421.052,174.200,26.090,154.578
C03296=1075.616,206.607,421.028,174.203,26.093,154.578
C03297=1075.621,206.855,421.003,174.205,26.096,154.578
C03298=1075.645,207.893,420.903,174.322,26.158,154.579
C03299=1075.655,208.304,420.861,174.325,26.164,154.579
C03300=1075.665,208.714,420.821,174.329,26.170,154.580
C03301=1075.675,209.125,420.780,174.332,26.176,154.581
C03302=1075.684,209.535,420.739,174.336,26.182,154.582
C03303=1075.690,209.784,420.715,174.338,26.186,154.583
C03304=1075.696,210.032,420.689,174.340,26.190,154.583
C03305=1075.701,210.281,420.665,174.342,26.194,154.584
C03306=1075.707,210.530,420.640,174.345,26.197,154.584
C03307=1075.712,210.779,420.615,174.347,26.201,154.585
C03308=1075.718,211.027,420.590,174.349,26.205,154.585
C03309=1075.724,211.277,420.565,174.351,26.209,154.586
C03310=1075.730,211.525,420.540,174.353,26.212,154.586
C03311=1075.736,211.773,420.515,174.356,26.216,154.587
C03312=1075.741,212.022,420.490,174.358,26.220,154.588
C03313=1075.747,212.270,420.465,174.360,26.224,154.588
C03314=1075.753,212.520,420.440,174.362,26.227,154.589
C03315=1075.758,212.768,420.415,174.364,26.231,154.589
C03316=1075.764,213.017,420.389,174.366,26.235,154.590
C03317=1075.770,213.266,420.365,174.369,26.238,154.590
C03318=1075.776,213.514,420.340,174.371,26.242,154.591
C03319=1075.782,213.763,420.315,174.373,26.246,154.591
C03320=1075.786,214.012,420.290,174.375,26.250,154.592
C03321=1075.793,214.260,420.264,174.377,26.253,154.592
C03322=1075.799,214.509,420.239,174.379,26.257,154.593
C03323=1075.804,214.757,420.215,174.382,26.261,154.594
C03324=1075.810,215.006,420.189,174.384,26.265,154.594
C03325=1075.816,215.255,420.163,174.386,26.268,154.595
C03326=1075.821,215.503,420.138,174.388,26.272,154.595
C03327=1075.827,215.753,420.113,174.390,26.276,154.596
C03328=1075.833,216.001,420.088,174.392,26.280,154.596
C03329=1075.838,216.249,420.063,174.395,26.283,154.597
C03330=1075.844,216.498,420.037,174.397,26.287,154.597
C03331=1075.850,216.747,420.012,174.399,26.290,154.598
C03332=1075.856,216.995,419.987,174.401,26.295,154.599
C03333=1075.862,217.244,419.962,174.403,26.298,154.599
C03334=1075.867,217.493,419.936,174.406,26.302,154.600
C03335=1075.873,217.742,419.911,174.408,26.305,154.600
C03336=1075.879,217.990,419.886,174.410,26.309,154.601
C03337=1075.884,218.239,419.860,174.412,26.313,154.601
C03338=1075.891,218.487,419.835,174.414,26.317,154.602
C03339=1075.897,218.736,419.809,174.417,26.320,154.602
C03340=1075.902,218.984,419.784,174.419,26.324,154.603
C03341=1075.908,219.233,419.758,174.421,26.328,154.603
C03342=1075.914,219.482,419.733,174.423,26.331,154.604
C03343=1075.919,219.731,419.708,174.425,26.335,154.604
C03344=1075.925,219.980,419.682,174.427,26.339,154.605
C03345=1075.930,220.228,419.657,174.430,26.342,154.606
C03346=1075.937,220.477,419.632,174.432,26.346,154.606
C03347=1075.943,220.726,419.606,174.434,26.350,154.607
C03348=1075.948,220.974,419.580,174.436,26.353,154.607
C03349=1075.955,221.223,419.554,174.439,26.357,154.608
C03350=1075.960,221.471,419.529,174.441,26.360,154.608
C03351=1075.970,221.886,419.486,174.445,26.367,154.609
C03352=1075.979,222.300,419.444,174.449,26.374,154.610
C03353=1075.989,222.715,419.401,174.453,26.379,154.611
C03354=1075.998,223.130,419.358,174.456,26.386,154.612
C03355=1076.004,223.378,419.333,174.458,26.389,154.612
C03356=1076.010,223.627,419.306,174.461,26.393,154.613
C03357=1076.015,223.876,419.280,174.463,26.397,154.613
C03358=1076.021,224.124,419.255,174.465,26.401,154.614
C03359=1076.026,224.373,419.229,174.467,26.404,154.614
C03360=1076.032,224.621,419.204,174.469,26.408,154.615
C03361=1076.038,224.870,419.177,174.472,26.412,154.616
C03362=1076.044,225.119,419.151,174.474,26.416,154.616
C03363=1076.050,225.367,419.126,174.476,26.419,154.617
C03364=1076.055,225.616,419.100,174.478,26.423,154.617
C03365=1076.062,225.864,419.074,174.481,26.427,154.618
C03366=1076.067,226.113,419.048,174.484,26.430,154.618
C03367=1076.072,226.362,419.022,174.486,26.434,154.619
C03368=1076.078,226.610,418.997,174.488,26.438,154.619
C03369=1076.084,226.859,418.970,174.490,26.442,154.620
C03370=1076.090,227.108,418.945,174.492,26.445,154.620
C03371=1076.096,227.356,418.919,174.495,26.449,154.621
C03372=1076.102,227.605,418.893,174.497,26.452,154.621
C03373=1076.107,227.854,418.867,174.499,26.456,154.622
C03374=1076.114,228.102,418.841,174.501,26.460,154.623
C03375=1076.119,228.351,418.815,174.503,26.464,154.623
C03376=1076.125,228.600,418.789,174.506,26.467,154.624
C03377=1076.131,228.848,418.763,174.509,26.471,154.624
C03378=1076.137,229.097,418.737,174.511,26.475,154.625
C03379=1076.142,229.345,418.710,174.513,26.478,154.625
C03380=1076.149,229.594,418.685,174.515,26.482,154.626
C03381=1076.154,229.842,418.658,174.518,26.485,154.626
C03382=1076.160,230.091,418.632,174.520,26.490,154.627
C03383=1076.166,230.339,418.606,174.522,26.493,154.627
C03384=1076.172,230.588,418.580,174.524,26.497,154.628
C03385=1076.178,230.836,418.554,174.527,26.500,154.628
C03386=1076.183,231.085,418.528,174.530,26.504,154.629
C03387=1076.189,231.334,418.501,174.532,26.508,154.630
C03388=1076.194,231.583,418.475,174.534,26.512,154.630
C03389=1076.200,231.831,418.448,174.536,26.516,154.631
C03390=1076.206,232.079,418.422,174.539,26.519,154.631
C03391=1076.212,232.328,418.396,174.541,26.523,154.632
C03392=1076.218,232.576,418.370,174.543,26.526,154.632
C03393=1076.223,232.825,418.344,174.545,26.530,154.633
C03394=1076.229,233.074,418.317,174.547,26.534,154.633
C03395=1076.235,233.322,418.291,174.551,26.538,154.634
C03396=1076.240,233.571,418.265,174.553,26.541,154.634
C03397=1076.246,233.820,418.238,174.555,26.545,154.635
C03398=1076.252,234.068,418.211,174.557,26.549,154.635
C03399=1076.258,234.316,418.185,174.559,26.553,154.636
C03400=1076.263,234.565,418.159,174.562,26.556,154.637
C03401=1076.269,234.814,418.132,174.564,26.560,154.637
C03402=1076.275,235.062,418.105,174.566,26.563,154.638
C03403=1076.284,235.468,418.062,174.571,26.570,154.639
C03404=1076.293,235.874,418.019,174.574,26.576,154.639
C03405=1076.303,236.281,417.976,174.578,26.582,154.640
C03406=1076.313,236.687,417.932,174.582,26.588,154.641
C03407=1076.318,236.935,417.905,174.584,26.592,154.642
C03408=1076.324,237.184,417.879,174.586,26.596,154.642
C03409=1076.329,237.433,417.852,174.588,26.599,154.643
C03410=1076.335,237.681,417.826,174.592,26.603,154.643
C03411=1076.341,237.930,417.799,174.594,26.607,154.644
C03412=1076.346,238.178,417.772,174.596,26.610,154.644
C03413=1076.352,238.426,417.746,174.598,26.614,154.645
C03414=1076.358,238.675,417.719,174.601,26.617,154.645
C03415=1076.364,238.924,417.692,174.603,26.621,154.646
C03416=1076.370,239.172,417.665,174.606,26.625,154.647
C03417=1076.376,239.421,417.639,174.608,26.629,154.647
C03418=1076.382,239.669,417.612,174.610,26.632,154.648
C03419=1076.387,239.917,417.585,174.613,26.636,154.648
C03420=1076.394,240.166,417.558,174.615,26.640,154.649
C03421=1076.399,240.415,417.531,174.617,26.644,154.649
C03422=1076.404,240.663,417.505,174.620,26.648,154.650
C03423=1076.410,240.912,417.478,174.623,26.651,154.650
C03424=1076.416,241.160,417.451,174.625,26.655,154.651
C03425=1076.422,241.409,417.424,174.627,26.658,154.651
C03426=1076.428,241.658,417.398,174.629,26.662,154.652
C03427=1076.434,241.906,417.371,174.632,26.665,154.652
C03428=1076.439,242.155,417.344,174.635,26.669,154.653
C03429=1076.445,242.402,417.316,174.637,26.673,154.654
C03430=1076.451,242.651,417.289,174.639,26.677,154.654
C03431=1076.457,242.900,417.263,174.641,26.681,154.655
C03432=1076.462,243.148,417.235,174.644,26.684,154.655
C03433=1076.468,243.397,417.209,174.647,26.688,154.656
C03434=1076.474,243.645,417.182,174.649,26.692,154.656
C03435=1076.480,243.894,417.154,174.651,26.696,154.657
C03436=1076.486,244.142,417.127,174.653,26.699,154.657
C03437=1076.491,244.391,417.101,174.656,26.703,154.658
C03438=1076.496,244.639,417.073,174.659,26.707,154.658
C03439=1076.503,244.888,417.046,174.661,26.711,154.659
C03440=1076.509,245.136,417.019,174.663,26.714,154.660
C03441=1076.514,245.385,416.992,174.666,26.718,154.660
C03442=1076.520,245.632,416.964,174.668,26.721,154.661
C03443=1076.526,245.882,416.937,174.671,26.726,154.661
C03444=1076.531,246.130,416.910,174.673,26.729,154.662
C03445=1076.537,246.378,416.883,174.675,26.733,154.662
C03446=1076.542,246.627,416.855,174.678,26.736,154.663
C03447=1076.549,246.876,416.828,174.680,26.740,154.663
C03448=1076.554,247.124,416.800,174.683,26.744,154.664
C03449=1076.560,247.372,416.774,174.685,26.748,154.664
C03450=1076.566,247.621,416.746,174.688,26.752,154.665
C03451=1076.572,247.869,416.719,174.690,26.755,154.666
C03452=1076.577,248.118,416.692,174.693,26.759,154.666
C03453=1076.583,248.366,416.664,174.695,26.763,154.667
C03454=1076.588,248.615,416.637,174.697,26.767,154.667
C03455=1076.597,249.014,416.592,174.701,26.773,154.668
C03456=1076.607,249.414,416.548,174.705,26.779,154.669
C03457=1076.616,249.814,416.504,174.710,26.785,154.670
C03458=1076.625,250.213,416.460,174.713,26.791,154.671
C03459=1076.631,250.461,416.432,174.716,26.795,154.671
C03460=1076.636,250.710,416.405,174.718,26.799,154.672
C03461=1076.642,250.958,416.377,174.721,26.802,154.672
C03462=1076.648,251.206,416.349,174.723,26.806,154.673
C03463=1076.653,251.455,416.322,174.725,26.810,154.674
C03464=1076.659,251.703,416.294,174.728,26.814,154.674
C03465=1076.665,251.952,416.267,174.731,26.817,154.675
C03466=1076.670,252.200,416.239,174.733,26.821,154.675
C03467=1076.676,252.448,416.211,174.735,26.825,154.676
C03468=1076.683,252.697,416.183,174.738,26.829,154.676
C03469=1076.688,252.946,416.156,174.741,26.832,154.677
C03470=1076.693,253.194,416.128,174.743,26.836,154.677
C03471=1076.700,253.442,416.100,174.745,26.840,154.678
C03472=1076.705,253.691,416.073,174.748,26.844,154.679
C03473=1076.711,253.940,416.045,174.751,26.847,154.679
C03474=1076.717,254.187,416.017,174.753,26.851,154.680
C03475=1076.723,254.436,415.989,174.755,26.855,154.680
C03476=1076.728,254.684,415.961,174.757,26.859,154.681
C03477=1076.734,254.932,415.934,174.761,26.862,154.681
C03478=1076.740,255.181,415.906,174.763,26.866,154.682
C03479=1076.745,255.429,415.878,174.765,26.870,154.682
C03480=1076.752,255.678,415.850,174.768,26.874,154.683
C03481=1076.757,255.926,415.822,174.771,26.877,154.683
C03482=1076.763,256.174,415.794,174.773,26.881,154.684
C03483=1076.768,256.423,415.766,174.775,26.885,154.685
C03484=1076.775,256.672,415.739,174.778,26.889,154.685
C03485=1076.780,256.920,415.711,174.781,26.892,154.686
C03486=1076.786,257.168,415.683,174.783,26.896,154.686
C03487=1076.791,257.416,415.655,174.786,26.900,154.687
C03488=1076.798,257.665,415.627,174.788,26.903,154.687
C03489=1076.803,257.913,415.599,174.790,26.907,154.688
C03490=1076.809,258.162,415.571,174.793,26.911,154.688
C03491=1076.815,258.410,415.543,174.796,26.915,154.689
C03492=1076.821,258.658,415.515,174.798,26.918,154.689
C03493=1076.827,258.907,415.487,174.801,26.922,154.690
C03494=1076.833,259.155,415.459,174.804,26.926,154.691
C03495=1076.839,259.404,415.431,174.806,26.930,154.691
C03496=1076.845,259.651,415.403,174.808,26.933,154.692
C03497=1076.851,259.900,415.375,174.811,26.937,154.692
C03498=1076.857,260.148,415.346,174.814,26.941,154.693
C03499=1076.862,260.396,415.318,174.816,26.944,154.693
C03500=1076.868,260.645,415.290,174.819,26.949,154.694
C03501=1076.875,260.894,415.262,174.821,26.952,154.694
C03502=1076.880,261.142,415.234,174.824,26.956,154.695
C03503=1076.886,261.390,415.206,174.827,26.960,154.695
C03504=1076.891,261.638,415.178,174.829,26.963,154.696
C03505=1076.898,261.887,415.149,174.832,26.967,154.696
C03506=1076.904,262.135,415.121,174.835,26.971,154.697
C03507=1076.913,262.532,415.075,174.838,26.977,154.698
C03508=1076.922,262.929,415.030,174.842,26.982,154.699
C03509=1076.932,263.326,414.985,174.847,26.988,154.700
C03510=1076.942,263.723,414.940,174.851,26.994,154.700
C03511=1076.948,263.971,414.911,174.853,26.998,154.701
C03512=1076.953,264.219,414.883,174.856,27.002,154.702
C03513=1076.960,264.467,414.854,174.859,27.005,154.702
C03514=1076.966,264.716,414.826,174.861,27.010,154.703
C03515=1076.971,264.964,414.798,174.864,27.013,154.703
C03516=1076.976,265.213,414.768,174.866,27.017,154.704
C03517=1076.982,265.461,414.740,174.869,27.021,154.704
C03518=1076.988,265.709,414.711,174.872,27.025,154.705
C03519=1076.994,265.958,414.683,174.874,27.028,154.705
C03520=1077.000,266.206,414.655,174.876,27.032,154.706
C03521=1077.006,266.454,414.626,174.880,27.036,154.707
C03522=1077.012,266.703,414.598,174.882,27.040,154.707
C03523=1077.018,266.951,414.569,174.884,27.044,154.708
C03524=1077.022,267.199,414.540,174.887,27.048,154.708
C03525=1077.029,267.447,414.511,174.890,27.051,154.709
C03526=1077.035,267.696,414.483,174.892,27.055,154.709
C03527=1077.041,267.944,414.454,174.895,27.059,154.710
C03528=1077.046,268.192,414.426,174.897,27.062,154.710
C03529=1077.052,268.440,414.397,174.901,27.066,154.711
C03530=1077.058,268.689,414.367,174.903,27.070,154.712
C03531=1077.064,268.937,414.339,174.905,27.074,154.712
C03532=1077.070,269.185,414.310,174.908,27.078,154.713
C03533=1077.075,269.434,414.282,174.910,27.082,154.713
C03534=1077.082,269.682,414.253,174.913,27.085,154.714
C03535=1077.087,269.930,414.223,174.916,27.089,154.714
C03536=1077.093,270.178,414.195,174.918,27.093,154.715
C03537=1077.099,270.426,414.166,174.921,27.097,154.716
C03538=1077.104,270.675,414.137,174.924,27.100,154.716
C03539=1077.111,270.923,414.108,174.926,27.104,154.717
C03540=1077.117,271.172,414.079,174.929,27.108,154.717
C03541=1077.122,271.419,414.051,174.931,27.112,154.718
C03542=1077.128,271.668,414.021,174.935,27.116,154.718
C03543=1077.134,271.916,413.992,174.937,27.120,154.719
C03544=1077.140,272.165,413.964,174.939,27.124,154.720
C03545=1077.145,272.413,413.934,174.942,27.127,154.720
C03546=1077.151,272.660,413.905,174.945,27.131,154.721
C03547=1077.157,272.909,413.876,174.948,27.135,154.721
C03548=1077.163,273.157,413.847,174.950,27.139,154.722
C03549=1077.169,273.406,413.818,174.952,27.142,154.722
C03550=1077.174,273.654,413.789,174.956,27.147,154.723
C03551=1077.180,273.902,413.760,174.958,27.150,154.723
C03552=1077.185,274.150,413.730,174.961,27.154,154.724
C03553=1077.192,274.398,413.701,174.963,27.158,154.725
C03554=1077.198,274.646,413.672,174.966,27.162,154.725
C03555=1077.203,274.895,413.643,174.969,27.166,154.726
C03556=1077.210,275.143,413.614,174.971,27.169,154.726
C03557=1077.215,275.391,413.584,174.974,27.174,154.727
C03558=1077.221,275.639,413.555,174.977,27.177,154.727
C03559=1077.230,276.040,413.508,174.981,27.184,154.728
C03560=1077.240,276.439,413.461,174.985,27.190,154.729
C03561=1077.249,276.840,413.413,174.990,27.196,154.730
C03562=1077.259,277.239,413.366,174.994,27.202,154.731
C03563=1077.264,277.487,413.336,174.997,27.206,154.732
C03564=1077.270,277.736,413.307,174.999,27.210,154.732
C03565=1077.276,277.984,413.278,175.002,27.214,154.733
C03566=1077.281,278.232,413.248,175.005,27.218,154.733
C03567=1077.288,278.481,413.219,175.008,27.222,154.734
C03568=1077.293,278.729,413.189,175.010,27.225,154.735
C03569=1077.299,278.977,413.160,175.012,27.229,154.735
C03570=1077.305,279.225,413.130,175.016,27.233,154.736
C03571=1077.311,279.473,413.100,175.018,27.237,154.736
C03572=1077.317,279.721,413.071,175.021,27.241,154.737
C03573=1077.322,279.970,413.041,175.023,27.245,154.738
C03574=1077.329,280.217,413.012,175.027,27.249,154.738
C03575=1077.335,280.466,412.982,175.029,27.252,154.739
C03576=1077.340,280.714,412.952,175.032,27.257,154.739
C03577=1077.346,280.962,412.923,175.034,27.260,154.740
C03578=1077.352,281.210,412.893,175.038,27.264,154.740
C03579=1077.358,281.459,412.863,175.040,27.268,154.741
C03580=1077.363,281.707,412.834,175.042,27.272,154.742
C03581=1077.369,281.955,412.803,175.045,27.276,154.742
C03582=1077.375,282.203,412.774,175.048,27.280,154.743
C03583=1077.381,282.451,412.744,175.051,27.284,154.743
C03584=1077.387,282.699,412.714,175.053,27.288,154.744
C03585=1077.392,282.948,412.685,175.056,27.292,154.745
C03586=1077.398,283.196,412.654,175.059,27.296,154.745
C03587=1077.404,283.444,412.625,175.062,27.300,154.746
C03588=1077.410,283.692,412.595,175.064,27.304,154.746
C03589=1077.415,283.940,412.565,175.067,27.307,154.747
C03590=1077.421,284.188,412.535,175.070,27.311,154.748
C03591=1077.427,284.436,412.505,175.073,27.315,154.748
C03592=1077.433,284.684,412.476,175.075,27.319,154.749
C03593=1077.439,284.932,412.446,175.078,27.324,154.749
C03594=1077.445,285.180,412.416,175.081,27.327,154.750
C03595=1077.450,285.429,412.386,175.084,27.331,154.751
C03596=1077.456,285.676,412.356,175.086,27.335,154.751
C03597=1077.462,285.925,412.325,175.089,27.339,154.752
C03598=1077.468,286.173,412.295,175.091,27.343,154.752
C03599=1077.474,286.421,412.266,175.095,27.347,154.753
C03600=1077.480,286.669,412.235,175.097,27.351,154.754
C03601=1077.486,286.917,412.206,175.100,27.355,154.754
C03602=1077.492,287.165,412.175,175.103,27.359,154.755
C03603=1077.497,287.413,412.145,175.106,27.362,154.755
C03604=1077.503,287.661,412.115,175.108,27.366,154.756
C03605=1077.509,287.910,412.085,175.111,27.371,154.757
C03606=1077.515,288.158,412.054,175.114,27.374,154.757
C03607=1077.521,288.406,412.025,175.117,27.379,154.758
C03608=1077.527,288.653,411.995,175.120,27.382,154.758
C03609=1077.533,288.901,411.964,175.122,27.386,154.759
C03610=1077.539,289.150,411.934,175.125,27.391,154.760
C03611=1077.548,289.559,411.884,175.129,27.397,154.761
C03612=1077.558,289.969,411.834,175.134,27.403,154.761
C03613=1077.567,290.380,411.784,175.139,27.410,154.763
C03614=1077.577,290.789,411.733,175.143,27.417,154.763
C03615=1077.584,291.038,411.703,175.147,27.421,154.764
C03616=1077.589,291.286,411.672,175.149,27.425,154.765
C03617=1077.595,291.534,411.642,175.152,27.429,154.765
C03618=1077.601,291.781,411.612,175.154,27.433,154.766
C03619=1077.607,292.029,411.581,175.158,27.437,154.767
C03620=1077.612,292.278,411.550,175.160,27.441,154.767
C03621=1077.618,292.526,411.520,175.163,27.445,154.768
C03622=1077.624,292.774,411.489,175.165,27.449,154.768
C03623=1077.630,293.022,411.459,175.169,27.453,154.769
C03624=1077.636,293.270,411.428,175.172,27.457,154.770
C03625=1077.642,293.518,411.398,175.174,27.461,154.770
C03626=1077.647,293.766,411.367,175.177,27.465,154.771
C03627=1077.653,294.014,411.337,175.180,27.469,154.772
C03628=1077.659,294.262,411.306,175.183,27.473,154.772
C03629=1077.665,294.510,411.276,175.185,27.477,154.773
C03630=1077.671,294.758,411.245,175.188,27.481,154.773
C03631=1077.678,295.006,411.214,175.192,27.485,154.774
C03632=1077.683,295.254,411.183,175.194,27.489,154.775
C03633=1077.689,295.502,411.152,175.197,27.493,154.775
C03634=1077.695,295.750,411.122,175.199,27.497,154.776
C03635=1077.701,295.998,411.091,175.203,27.501,154.776
C03636=1077.706,296.246,411.060,175.206,27.506,154.777
C03637=1077.713,296.494,411.029,175.208,27.509,154.778
C03638=1077.719,296.742,410.999,175.211,27.514,154.778
C03639=1077.724,296.990,410.968,175.214,27.517,154.779
C03640=1077.730,297.238,410.936,175.217,27.521,154.780
